//=============================================================================
// ST10_Flow7_CGlueing.scl
// 1:1 CONVERSION FROM TIA PORTAL V18 GRAPH XML
// Generated: 2026-02-02
//=============================================================================

TYPE
    E_STEP_ST10_Flow7_CGlueing : (
        STEP_ST10_Flow7_CGlueing_JudgeYPosition := 90,
        STEP_ST10_Flow7_CGlueing_CameraCheck1 := 118,
        STEP_ST10_Flow7_CGlueing_Step161 := 161,
        STEP_ST10_Flow7_CGlueing_Servo_returns_toGluePos_4 := 56,
        STEP_ST10_Flow7_CGlueing_OKStatus_3 := 135,
        STEP_ST10_Flow7_CGlueing_MESOverTime_1 := 318,
        STEP_ST10_Flow7_CGlueing_Axis_YToGlueePos_5 := 41,
        STEP_ST10_Flow7_CGlueing_ShaftGlueCameraCheck := 250,
        STEP_ST10_Flow7_CGlueing_CheckGlueSysOK_4 := 72,
        STEP_ST10_Flow7_CGlueing_ResetMesCheckRequest_1 := 302,
        STEP_ST10_Flow7_CGlueing_ServoHomePos_5 := 143,
        STEP_ST10_Flow7_CGlueing_MES_Check := 150,
        STEP_ST10_Flow7_CGlueing_Axis_XToGluePos_6 := 92,
        STEP_ST10_Flow7_CGlueing_Axis_ZToGlueePos_6 := 93,
        STEP_ST10_Flow7_CGlueing_CameraCheck4 := 137,
        STEP_ST10_Flow7_CGlueing_CheckIV3Ready_3 := 207,
        STEP_ST10_Flow7_CGlueing_Axis_XToGluePos_4 := 54,
        STEP_ST10_Flow7_CGlueing_GluePos_2 := 98,
        STEP_ST10_Flow7_CGlueing_OKStatus_4 := 141,
        STEP_ST10_Flow7_CGlueing_GlueFinishStatus := 83,
        STEP_ST10_Flow7_CGlueing_Axis_XToGluePos_5 := 71,
        STEP_ST10_Flow7_CGlueing_IAIMoveFinish_1 := 105,
        STEP_ST10_Flow7_CGlueing_MESOverTime := 323,
        STEP_ST10_Flow7_CGlueing_Axis_YToGluePos_6 := 91,
        STEP_ST10_Flow7_CGlueing_CheckServo_returns_toHome_Pos_5 := 99,
        STEP_ST10_Flow7_CGlueing_Step104 := 104,
        STEP_ST10_Flow7_CGlueing_OKStatus_2 := 129,
        STEP_ST10_Flow7_CGlueing_StatusAlarm := 24,
        STEP_ST10_Flow7_CGlueing_IV3Check_2 := 127,
        STEP_ST10_Flow7_CGlueing_WaitRobotFinishTask_2 := 289,
        STEP_ST10_Flow7_CGlueing_JudgeCheckStatus_3 := 134,
        STEP_ST10_Flow7_CGlueing_Axis_XToGluePos_2 := 36,
        STEP_ST10_Flow7_CGlueing_Axis_XToGlueSafPos_4 := 57,
        STEP_ST10_Flow7_CGlueing_PutMagnet := 64,
        STEP_ST10_Flow7_CGlueing_NGStatus_4 := 142,
        STEP_ST10_Flow7_CGlueing_F7_Initial := 1,
        STEP_ST10_Flow7_CGlueing_ok := 311,
        STEP_ST10_Flow7_CGlueing_Axis_ZToGlueePos_7 := 148,
        STEP_ST10_Flow7_CGlueing_CheckGlueSysOK_1 := 37,
        STEP_ST10_Flow7_CGlueing_ServoJoging := 123,
        STEP_ST10_Flow7_CGlueing_IAIMoveFinish_3 := 111,
        STEP_ST10_Flow7_CGlueing_RobotGluePick := 400,
        STEP_ST10_Flow7_CGlueing_C_LocationCylinderToHP2 := 122,
        STEP_ST10_Flow7_CGlueing_CheckIV3Ready_1 := 204,
        STEP_ST10_Flow7_CGlueing_Glue_3 := 50,
        STEP_ST10_Flow7_CGlueing_MES_Check_OK := 306,
        STEP_ST10_Flow7_CGlueing_Prepare_MES_CheckData := 303,
        STEP_ST10_Flow7_CGlueing_ServoHomePos_1 := 97,
        STEP_ST10_Flow7_CGlueing_Shaft_Glue := 287,
        STEP_ST10_Flow7_CGlueing_JudgeCheckStatus_4 := 140,
        STEP_ST10_Flow7_CGlueing_MESSaveRequest_1 := 313,
        STEP_ST10_Flow7_CGlueing_Axis_XYToHomePos_1 := 86,
        STEP_ST10_Flow7_CGlueing_JudgeCheckStatus := 61,
        STEP_ST10_Flow7_CGlueing_CameraCheck3 := 131,
        STEP_ST10_Flow7_CGlueing_Axis_ZToHomePos_2 := 82,
        STEP_ST10_Flow7_CGlueing_RequestRobotPutMagnet_1 := 281,
        STEP_ST10_Flow7_CGlueing_MESResult := 151,
        STEP_ST10_Flow7_CGlueing_CheckIV3Ready := 202,
        STEP_ST10_Flow7_CGlueing_MES__Check_Result := 350,
        STEP_ST10_Flow7_CGlueing_StopServoJoging := 124,
        STEP_ST10_Flow7_CGlueing_NGStatus := 63,
        STEP_ST10_Flow7_CGlueing_OKPart := 152,
        STEP_ST10_Flow7_CGlueing_IAIMoveFinish := 95,
        STEP_ST10_Flow7_CGlueing_Step159 := 159,
        STEP_ST10_Flow7_CGlueing_Step160 := 160,
        STEP_ST10_Flow7_CGlueing_Servo_returns_toGluePos_8 := 138,
        STEP_ST10_Flow7_CGlueing_Axis_YToGlueePos_1 := 26,
        STEP_ST10_Flow7_CGlueing_S10_InitialFinish := 10,
        STEP_ST10_Flow7_CGlueing_CheckIV3Ready_2 := 206,
        STEP_ST10_Flow7_CGlueing_Check_OK := 316,
        STEP_ST10_Flow7_CGlueing_NGStatus_3 := 136,
        STEP_ST10_Flow7_CGlueing_GluePos_1 := 96,
        STEP_ST10_Flow7_CGlueing_PartNG := 401,
        STEP_ST10_Flow7_CGlueing_JudgeCheckStatus_2 := 128,
        STEP_ST10_Flow7_CGlueing_RequestRobot1PutShaft := 27,
        STEP_ST10_Flow7_CGlueing_MES_Check_OK_1 := 399,
        STEP_ST10_Flow7_CGlueing_Process_Finish := 149,
        STEP_ST10_Flow7_CGlueing_Shaft_GlueCheck := 67,
        STEP_ST10_Flow7_CGlueing_ServoReady_ := 6,
        STEP_ST10_Flow7_CGlueing_MagnetGlueFinish := 349,
        STEP_ST10_Flow7_CGlueing_WaitRobotFinishTask_1 := 288,
        STEP_ST10_Flow7_CGlueing_Glue_2 := 40,
        STEP_ST10_Flow7_CGlueing_Bypass_1 := 324,
        STEP_ST10_Flow7_CGlueing_Step314 := 322,
        STEP_ST10_Flow7_CGlueing_Axis_ZToGlueePos_5 := 70,
        STEP_ST10_Flow7_CGlueing_IV3Check_1 := 69,
        STEP_ST10_Flow7_CGlueing_Step102 := 102,
        STEP_ST10_Flow7_CGlueing_Axis_YToGlueePos_7 := 88,
        STEP_ST10_Flow7_CGlueing_Servo_returns_toGluePos_2 := 38,
        STEP_ST10_Flow7_CGlueing_Axis_XToGluePos_3 := 46,
        STEP_ST10_Flow7_CGlueing_S4 := 4,
        STEP_ST10_Flow7_CGlueing_C_LocationCylinderToWP_1 := 120,
        STEP_ST10_Flow7_CGlueing_IAIMoveFinish__1 := 153,
        STEP_ST10_Flow7_CGlueing_JudgeCheckStatus_1 := 74,
        STEP_ST10_Flow7_CGlueing_Axis_ZToHomePos_1 := 80,
        STEP_ST10_Flow7_CGlueing_GluePos_4 := 116,
        STEP_ST10_Flow7_CGlueing_Axis_XToGlueSafPos_3 := 49,
        STEP_ST10_Flow7_CGlueing_ShaftGlueFinishStatus := 68,
        STEP_ST10_Flow7_CGlueing_Servo_returns_toGluePos_6 := 125,
        STEP_ST10_Flow7_CGlueing_Axis_XToHomePos := 81,
        STEP_ST10_Flow7_CGlueing_Step87 := 87,
        STEP_ST10_Flow7_CGlueing_Step315 := 328,
        STEP_ST10_Flow7_CGlueing_CheckPartStatus := 23,
        STEP_ST10_Flow7_CGlueing_Step158 := 158,
        STEP_ST10_Flow7_CGlueing_WaitIAIStop := 103,
        STEP_ST10_Flow7_CGlueing_Axis_ZToGlueePos_3 := 45,
        STEP_ST10_Flow7_CGlueing_CheckGlueSysOK_3 := 55,
        STEP_ST10_Flow7_CGlueing_WaitTableCode_OK := 101,
        STEP_ST10_Flow7_CGlueing_Axis_YToGlueePos_6 := 52,
        STEP_ST10_Flow7_CGlueing_NGStatus_1 := 85,
        STEP_ST10_Flow7_CGlueing_GluePos_3 := 114,
        STEP_ST10_Flow7_CGlueing_Step146 := 146,
        STEP_ST10_Flow7_CGlueing_Axis_XYToHomePos_2 := 156,
        STEP_ST10_Flow7_CGlueing_S3 := 3,
        STEP_ST10_Flow7_CGlueing_ServoHomePos_2 := 113,
        STEP_ST10_Flow7_CGlueing_Servo_returns_toGluePos_5 := 73,
        STEP_ST10_Flow7_CGlueing_ResetMesCheckRequest := 301,
        STEP_ST10_Flow7_CGlueing_Axis_XYIVCheckPos := 79,
        STEP_ST10_Flow7_CGlueing_OKStatus := 62,
        STEP_ST10_Flow7_CGlueing_S5_MESInitial := 5,
        STEP_ST10_Flow7_CGlueing_ShaftGluingProcess := 200,
        STEP_ST10_Flow7_CGlueing_Axis_ZToGlueePos_4 := 53,
        STEP_ST10_Flow7_CGlueing_CheckGlueSysOK_2 := 47,
        STEP_ST10_Flow7_CGlueing_RobotPutMagnet := 300,
        STEP_ST10_Flow7_CGlueing_TimeDelay_4 := 59,
        STEP_ST10_Flow7_CGlueing_Axis_XYIVCheckPos_1 := 157,
        STEP_ST10_Flow7_CGlueing_Axis_YToGluePos_5 := 75,
        STEP_ST10_Flow7_CGlueing_C_LocationCylinderToWP_2 := 121,
        STEP_ST10_Flow7_CGlueing_ServoHomePos_4 := 117,
        STEP_ST10_Flow7_CGlueing_Servo_returns_toGluePos_1 := 31,
        STEP_ST10_Flow7_CGlueing_ProcessStart := 100,
        STEP_ST10_Flow7_CGlueing_Servo_returns_toGluePos_7 := 132,
        STEP_ST10_Flow7_CGlueing_Axis_XToGlueSafPos_2 := 39,
        STEP_ST10_Flow7_CGlueing_TimeDelay_3 := 51,
        STEP_ST10_Flow7_CGlueing_ServoHomePos_6 := 144,
        STEP_ST10_Flow7_CGlueing_RequestRobotGluePick := 282,
        STEP_ST10_Flow7_CGlueing_MESCheckRequest := 310,
        STEP_ST10_Flow7_CGlueing_Axis_ZToIVCheckPos := 78,
        STEP_ST10_Flow7_CGlueing_ok_1 := 329,
        STEP_ST10_Flow7_CGlueing_CheckGlueSysOK := 30,
        STEP_ST10_Flow7_CGlueing_IAIMoveFinish_2 := 108,
        STEP_ST10_Flow7_CGlueing_Axis_ZToGlueePos_1 := 89,
        STEP_ST10_Flow7_CGlueing_Glue2s := 163,
        STEP_ST10_Flow7_CGlueing_ServoHomePos := 94,
        STEP_ST10_Flow7_CGlueing_Axis_ZToGlueePos_2 := 35,
        STEP_ST10_Flow7_CGlueing_IV3Check := 60,
        STEP_ST10_Flow7_CGlueing_Step110 := 110,
        STEP_ST10_Flow7_CGlueing_Magnet_Glue := 65,
        STEP_ST10_Flow7_CGlueing_Servo_returns_toGluePos_3 := 48,
        STEP_ST10_Flow7_CGlueing_WaitIAIStop_3 := 112,
        STEP_ST10_Flow7_CGlueing_ResultNG := 326,
        STEP_ST10_Flow7_CGlueing_NGStatus_2 := 130,
        STEP_ST10_Flow7_CGlueing_TimeDelay_1 := 42,
        STEP_ST10_Flow7_CGlueing_Bypass := 315,
        STEP_ST10_Flow7_CGlueing_IAIMoveFinish_4 := 155,
        STEP_ST10_Flow7_CGlueing_CheckIV3Ready_4 := 208,
        STEP_ST10_Flow7_CGlueing_ShaftGlueProcessFinish := 299,
        STEP_ST10_Flow7_CGlueing_WaitIAIStop_1 := 106,
        STEP_ST10_Flow7_CGlueing_Check_NG := 317,
        STEP_ST10_Flow7_CGlueing_TimeDelay_5 := 76,
        STEP_ST10_Flow7_CGlueing_Servo_returns_toHome_Pos := 22,
        STEP_ST10_Flow7_CGlueing_ServoHomePos_3 := 115,
        STEP_ST10_Flow7_CGlueing_CameraCheck2 := 126,
        STEP_ST10_Flow7_CGlueing_WaitRobot1FinishTask := 28,
        STEP_ST10_Flow7_CGlueing_bypassGlue4 := 162,
        STEP_ST10_Flow7_CGlueing_IV3Check_4 := 139,
        STEP_ST10_Flow7_CGlueing_IV3_Check := 630,
        STEP_ST10_Flow7_CGlueing_Prepare_MES_CheckData_1 := 307,
        STEP_ST10_Flow7_CGlueing_MaganetGlue := 320,
        STEP_ST10_Flow7_CGlueing_WaitIAIStop_2 := 109,
        STEP_ST10_Flow7_CGlueing_Axis_XToGlueSafPos := 32,
        STEP_ST10_Flow7_CGlueing_IAIMoveFinish_5 := 154,
        STEP_ST10_Flow7_CGlueing_Total_Score_of_Shaft_Gluening_check := 203,
        STEP_ST10_Flow7_CGlueing_Axis_YToHomePos := 21,
        STEP_ST10_Flow7_CGlueing_TimeDelay_2 := 43,
        STEP_ST10_Flow7_CGlueing_Step145 := 145,
        STEP_ST10_Flow7_CGlueing_CheckAxisXPos := 147,
        STEP_ST10_Flow7_CGlueing_C_LocationCylinderToHP := 119,
        STEP_ST10_Flow7_CGlueing_OKStatus_1 := 84,
        STEP_ST10_Flow7_CGlueing_Step204 := 205,
        STEP_ST10_Flow7_CGlueing_Step107 := 107,
        STEP_ST10_Flow7_CGlueing_Process__Finish := 290,
        STEP_ST10_Flow7_CGlueing_Glue_4 := 58,
        STEP_ST10_Flow7_CGlueing_Glue_1 := 33,
        STEP_ST10_Flow7_CGlueing_IV3Check_3 := 133,
        STEP_ST10_Flow7_CGlueing_Magnet_GlueCheck := 66,
        STEP_ST10_Flow7_CGlueing_WaitRobotInitialFinish := 8,
        STEP_ST10_Flow7_CGlueing_S2 := 2,
        STEP_ST10_Flow7_CGlueing_Axis_XToGluePos_1 := 29,
    ) INT := 1;
END_TYPE

CONST
    STEP_ST10_Flow7_CGlueing_JudgeYPosition := 90;
    STEP_ST10_Flow7_CGlueing_CameraCheck1 := 118;
    STEP_ST10_Flow7_CGlueing_Step161 := 161;
    STEP_ST10_Flow7_CGlueing_Servo_returns_toGluePos_4 := 56;
    STEP_ST10_Flow7_CGlueing_OKStatus_3 := 135;
    STEP_ST10_Flow7_CGlueing_MESOverTime_1 := 318;
    STEP_ST10_Flow7_CGlueing_Axis_YToGlueePos_5 := 41;
    STEP_ST10_Flow7_CGlueing_ShaftGlueCameraCheck := 250;
    STEP_ST10_Flow7_CGlueing_CheckGlueSysOK_4 := 72;
    STEP_ST10_Flow7_CGlueing_ResetMesCheckRequest_1 := 302;
    STEP_ST10_Flow7_CGlueing_ServoHomePos_5 := 143;
    STEP_ST10_Flow7_CGlueing_MES_Check := 150;
    STEP_ST10_Flow7_CGlueing_Axis_XToGluePos_6 := 92;
    STEP_ST10_Flow7_CGlueing_Axis_ZToGlueePos_6 := 93;
    STEP_ST10_Flow7_CGlueing_CameraCheck4 := 137;
    STEP_ST10_Flow7_CGlueing_CheckIV3Ready_3 := 207;
    STEP_ST10_Flow7_CGlueing_Axis_XToGluePos_4 := 54;
    STEP_ST10_Flow7_CGlueing_GluePos_2 := 98;
    STEP_ST10_Flow7_CGlueing_OKStatus_4 := 141;
    STEP_ST10_Flow7_CGlueing_GlueFinishStatus := 83;
    STEP_ST10_Flow7_CGlueing_Axis_XToGluePos_5 := 71;
    STEP_ST10_Flow7_CGlueing_IAIMoveFinish_1 := 105;
    STEP_ST10_Flow7_CGlueing_MESOverTime := 323;
    STEP_ST10_Flow7_CGlueing_Axis_YToGluePos_6 := 91;
    STEP_ST10_Flow7_CGlueing_CheckServo_returns_toHome_Pos_5 := 99;
    STEP_ST10_Flow7_CGlueing_Step104 := 104;
    STEP_ST10_Flow7_CGlueing_OKStatus_2 := 129;
    STEP_ST10_Flow7_CGlueing_StatusAlarm := 24;
    STEP_ST10_Flow7_CGlueing_IV3Check_2 := 127;
    STEP_ST10_Flow7_CGlueing_WaitRobotFinishTask_2 := 289;
    STEP_ST10_Flow7_CGlueing_JudgeCheckStatus_3 := 134;
    STEP_ST10_Flow7_CGlueing_Axis_XToGluePos_2 := 36;
    STEP_ST10_Flow7_CGlueing_Axis_XToGlueSafPos_4 := 57;
    STEP_ST10_Flow7_CGlueing_PutMagnet := 64;
    STEP_ST10_Flow7_CGlueing_NGStatus_4 := 142;
    STEP_ST10_Flow7_CGlueing_F7_Initial := 1;
    STEP_ST10_Flow7_CGlueing_ok := 311;
    STEP_ST10_Flow7_CGlueing_Axis_ZToGlueePos_7 := 148;
    STEP_ST10_Flow7_CGlueing_CheckGlueSysOK_1 := 37;
    STEP_ST10_Flow7_CGlueing_ServoJoging := 123;
    STEP_ST10_Flow7_CGlueing_IAIMoveFinish_3 := 111;
    STEP_ST10_Flow7_CGlueing_RobotGluePick := 400;
    STEP_ST10_Flow7_CGlueing_C_LocationCylinderToHP2 := 122;
    STEP_ST10_Flow7_CGlueing_CheckIV3Ready_1 := 204;
    STEP_ST10_Flow7_CGlueing_Glue_3 := 50;
    STEP_ST10_Flow7_CGlueing_MES_Check_OK := 306;
    STEP_ST10_Flow7_CGlueing_Prepare_MES_CheckData := 303;
    STEP_ST10_Flow7_CGlueing_ServoHomePos_1 := 97;
    STEP_ST10_Flow7_CGlueing_Shaft_Glue := 287;
    STEP_ST10_Flow7_CGlueing_JudgeCheckStatus_4 := 140;
    STEP_ST10_Flow7_CGlueing_MESSaveRequest_1 := 313;
    STEP_ST10_Flow7_CGlueing_Axis_XYToHomePos_1 := 86;
    STEP_ST10_Flow7_CGlueing_JudgeCheckStatus := 61;
    STEP_ST10_Flow7_CGlueing_CameraCheck3 := 131;
    STEP_ST10_Flow7_CGlueing_Axis_ZToHomePos_2 := 82;
    STEP_ST10_Flow7_CGlueing_RequestRobotPutMagnet_1 := 281;
    STEP_ST10_Flow7_CGlueing_MESResult := 151;
    STEP_ST10_Flow7_CGlueing_CheckIV3Ready := 202;
    STEP_ST10_Flow7_CGlueing_MES__Check_Result := 350;
    STEP_ST10_Flow7_CGlueing_StopServoJoging := 124;
    STEP_ST10_Flow7_CGlueing_NGStatus := 63;
    STEP_ST10_Flow7_CGlueing_OKPart := 152;
    STEP_ST10_Flow7_CGlueing_IAIMoveFinish := 95;
    STEP_ST10_Flow7_CGlueing_Step159 := 159;
    STEP_ST10_Flow7_CGlueing_Step160 := 160;
    STEP_ST10_Flow7_CGlueing_Servo_returns_toGluePos_8 := 138;
    STEP_ST10_Flow7_CGlueing_Axis_YToGlueePos_1 := 26;
    STEP_ST10_Flow7_CGlueing_S10_InitialFinish := 10;
    STEP_ST10_Flow7_CGlueing_CheckIV3Ready_2 := 206;
    STEP_ST10_Flow7_CGlueing_Check_OK := 316;
    STEP_ST10_Flow7_CGlueing_NGStatus_3 := 136;
    STEP_ST10_Flow7_CGlueing_GluePos_1 := 96;
    STEP_ST10_Flow7_CGlueing_PartNG := 401;
    STEP_ST10_Flow7_CGlueing_JudgeCheckStatus_2 := 128;
    STEP_ST10_Flow7_CGlueing_RequestRobot1PutShaft := 27;
    STEP_ST10_Flow7_CGlueing_MES_Check_OK_1 := 399;
    STEP_ST10_Flow7_CGlueing_Process_Finish := 149;
    STEP_ST10_Flow7_CGlueing_Shaft_GlueCheck := 67;
    STEP_ST10_Flow7_CGlueing_ServoReady_ := 6;
    STEP_ST10_Flow7_CGlueing_MagnetGlueFinish := 349;
    STEP_ST10_Flow7_CGlueing_WaitRobotFinishTask_1 := 288;
    STEP_ST10_Flow7_CGlueing_Glue_2 := 40;
    STEP_ST10_Flow7_CGlueing_Bypass_1 := 324;
    STEP_ST10_Flow7_CGlueing_Step314 := 322;
    STEP_ST10_Flow7_CGlueing_Axis_ZToGlueePos_5 := 70;
    STEP_ST10_Flow7_CGlueing_IV3Check_1 := 69;
    STEP_ST10_Flow7_CGlueing_Step102 := 102;
    STEP_ST10_Flow7_CGlueing_Axis_YToGlueePos_7 := 88;
    STEP_ST10_Flow7_CGlueing_Servo_returns_toGluePos_2 := 38;
    STEP_ST10_Flow7_CGlueing_Axis_XToGluePos_3 := 46;
    STEP_ST10_Flow7_CGlueing_S4 := 4;
    STEP_ST10_Flow7_CGlueing_C_LocationCylinderToWP_1 := 120;
    STEP_ST10_Flow7_CGlueing_IAIMoveFinish__1 := 153;
    STEP_ST10_Flow7_CGlueing_JudgeCheckStatus_1 := 74;
    STEP_ST10_Flow7_CGlueing_Axis_ZToHomePos_1 := 80;
    STEP_ST10_Flow7_CGlueing_GluePos_4 := 116;
    STEP_ST10_Flow7_CGlueing_Axis_XToGlueSafPos_3 := 49;
    STEP_ST10_Flow7_CGlueing_ShaftGlueFinishStatus := 68;
    STEP_ST10_Flow7_CGlueing_Servo_returns_toGluePos_6 := 125;
    STEP_ST10_Flow7_CGlueing_Axis_XToHomePos := 81;
    STEP_ST10_Flow7_CGlueing_Step87 := 87;
    STEP_ST10_Flow7_CGlueing_Step315 := 328;
    STEP_ST10_Flow7_CGlueing_CheckPartStatus := 23;
    STEP_ST10_Flow7_CGlueing_Step158 := 158;
    STEP_ST10_Flow7_CGlueing_WaitIAIStop := 103;
    STEP_ST10_Flow7_CGlueing_Axis_ZToGlueePos_3 := 45;
    STEP_ST10_Flow7_CGlueing_CheckGlueSysOK_3 := 55;
    STEP_ST10_Flow7_CGlueing_WaitTableCode_OK := 101;
    STEP_ST10_Flow7_CGlueing_Axis_YToGlueePos_6 := 52;
    STEP_ST10_Flow7_CGlueing_NGStatus_1 := 85;
    STEP_ST10_Flow7_CGlueing_GluePos_3 := 114;
    STEP_ST10_Flow7_CGlueing_Step146 := 146;
    STEP_ST10_Flow7_CGlueing_Axis_XYToHomePos_2 := 156;
    STEP_ST10_Flow7_CGlueing_S3 := 3;
    STEP_ST10_Flow7_CGlueing_ServoHomePos_2 := 113;
    STEP_ST10_Flow7_CGlueing_Servo_returns_toGluePos_5 := 73;
    STEP_ST10_Flow7_CGlueing_ResetMesCheckRequest := 301;
    STEP_ST10_Flow7_CGlueing_Axis_XYIVCheckPos := 79;
    STEP_ST10_Flow7_CGlueing_OKStatus := 62;
    STEP_ST10_Flow7_CGlueing_S5_MESInitial := 5;
    STEP_ST10_Flow7_CGlueing_ShaftGluingProcess := 200;
    STEP_ST10_Flow7_CGlueing_Axis_ZToGlueePos_4 := 53;
    STEP_ST10_Flow7_CGlueing_CheckGlueSysOK_2 := 47;
    STEP_ST10_Flow7_CGlueing_RobotPutMagnet := 300;
    STEP_ST10_Flow7_CGlueing_TimeDelay_4 := 59;
    STEP_ST10_Flow7_CGlueing_Axis_XYIVCheckPos_1 := 157;
    STEP_ST10_Flow7_CGlueing_Axis_YToGluePos_5 := 75;
    STEP_ST10_Flow7_CGlueing_C_LocationCylinderToWP_2 := 121;
    STEP_ST10_Flow7_CGlueing_ServoHomePos_4 := 117;
    STEP_ST10_Flow7_CGlueing_Servo_returns_toGluePos_1 := 31;
    STEP_ST10_Flow7_CGlueing_ProcessStart := 100;
    STEP_ST10_Flow7_CGlueing_Servo_returns_toGluePos_7 := 132;
    STEP_ST10_Flow7_CGlueing_Axis_XToGlueSafPos_2 := 39;
    STEP_ST10_Flow7_CGlueing_TimeDelay_3 := 51;
    STEP_ST10_Flow7_CGlueing_ServoHomePos_6 := 144;
    STEP_ST10_Flow7_CGlueing_RequestRobotGluePick := 282;
    STEP_ST10_Flow7_CGlueing_MESCheckRequest := 310;
    STEP_ST10_Flow7_CGlueing_Axis_ZToIVCheckPos := 78;
    STEP_ST10_Flow7_CGlueing_ok_1 := 329;
    STEP_ST10_Flow7_CGlueing_CheckGlueSysOK := 30;
    STEP_ST10_Flow7_CGlueing_IAIMoveFinish_2 := 108;
    STEP_ST10_Flow7_CGlueing_Axis_ZToGlueePos_1 := 89;
    STEP_ST10_Flow7_CGlueing_Glue2s := 163;
    STEP_ST10_Flow7_CGlueing_ServoHomePos := 94;
    STEP_ST10_Flow7_CGlueing_Axis_ZToGlueePos_2 := 35;
    STEP_ST10_Flow7_CGlueing_IV3Check := 60;
    STEP_ST10_Flow7_CGlueing_Step110 := 110;
    STEP_ST10_Flow7_CGlueing_Magnet_Glue := 65;
    STEP_ST10_Flow7_CGlueing_Servo_returns_toGluePos_3 := 48;
    STEP_ST10_Flow7_CGlueing_WaitIAIStop_3 := 112;
    STEP_ST10_Flow7_CGlueing_ResultNG := 326;
    STEP_ST10_Flow7_CGlueing_NGStatus_2 := 130;
    STEP_ST10_Flow7_CGlueing_TimeDelay_1 := 42;
    STEP_ST10_Flow7_CGlueing_Bypass := 315;
    STEP_ST10_Flow7_CGlueing_IAIMoveFinish_4 := 155;
    STEP_ST10_Flow7_CGlueing_CheckIV3Ready_4 := 208;
    STEP_ST10_Flow7_CGlueing_ShaftGlueProcessFinish := 299;
    STEP_ST10_Flow7_CGlueing_WaitIAIStop_1 := 106;
    STEP_ST10_Flow7_CGlueing_Check_NG := 317;
    STEP_ST10_Flow7_CGlueing_TimeDelay_5 := 76;
    STEP_ST10_Flow7_CGlueing_Servo_returns_toHome_Pos := 22;
    STEP_ST10_Flow7_CGlueing_ServoHomePos_3 := 115;
    STEP_ST10_Flow7_CGlueing_CameraCheck2 := 126;
    STEP_ST10_Flow7_CGlueing_WaitRobot1FinishTask := 28;
    STEP_ST10_Flow7_CGlueing_bypassGlue4 := 162;
    STEP_ST10_Flow7_CGlueing_IV3Check_4 := 139;
    STEP_ST10_Flow7_CGlueing_IV3_Check := 630;
    STEP_ST10_Flow7_CGlueing_Prepare_MES_CheckData_1 := 307;
    STEP_ST10_Flow7_CGlueing_MaganetGlue := 320;
    STEP_ST10_Flow7_CGlueing_WaitIAIStop_2 := 109;
    STEP_ST10_Flow7_CGlueing_Axis_XToGlueSafPos := 32;
    STEP_ST10_Flow7_CGlueing_IAIMoveFinish_5 := 154;
    STEP_ST10_Flow7_CGlueing_Total_Score_of_Shaft_Gluening_check := 203;
    STEP_ST10_Flow7_CGlueing_Axis_YToHomePos := 21;
    STEP_ST10_Flow7_CGlueing_TimeDelay_2 := 43;
    STEP_ST10_Flow7_CGlueing_Step145 := 145;
    STEP_ST10_Flow7_CGlueing_CheckAxisXPos := 147;
    STEP_ST10_Flow7_CGlueing_C_LocationCylinderToHP := 119;
    STEP_ST10_Flow7_CGlueing_OKStatus_1 := 84;
    STEP_ST10_Flow7_CGlueing_Step204 := 205;
    STEP_ST10_Flow7_CGlueing_Step107 := 107;
    STEP_ST10_Flow7_CGlueing_Process__Finish := 290;
    STEP_ST10_Flow7_CGlueing_Glue_4 := 58;
    STEP_ST10_Flow7_CGlueing_Glue_1 := 33;
    STEP_ST10_Flow7_CGlueing_IV3Check_3 := 133;
    STEP_ST10_Flow7_CGlueing_Magnet_GlueCheck := 66;
    STEP_ST10_Flow7_CGlueing_WaitRobotInitialFinish := 8;
    STEP_ST10_Flow7_CGlueing_S2 := 2;
    STEP_ST10_Flow7_CGlueing_Axis_XToGluePos_1 := 29;
END_CONST

FUNCTION_BLOCK "ST10_Flow7_CGlueing_1to1"
{ S7_Optimized_Access := 'TRUE' }
VERSION : 1.0

VAR_INPUT
    iSysInface : "RCS_SysComInterface_V1";
END_VAR

VAR_IN_OUT
    ioPM_Inface : "RCS_PMInterface_V1";
    ioStatus : Int;
END_VAR

VAR_OUTPUT
    oAlarmID : Int;
END_VAR

VAR
    State : INT := 1;
    act_InitialRun : Bool;
    act_InitialOK : Bool;
    act_WaitRunning : Bool;
    act_Running : Bool;
    act_ProcessComplete : Bool;
    act_ProcessStart : Bool;
    act_UnPause : Bool;
    bError : Bool;
    wErrorID : Word;
END_VAR

BEGIN
    //======================================================================
    // STATE MACHINE - Inline Transition Conditions
    //======================================================================

    CASE #State OF

        // ===========================================
        // STEP 90: JudgeYPosition
        // ===========================================
        STEP_ST10_Flow7_CGlueing_JudgeYPosition:
            // No actions in XML

            // Transition to next step: 118
            IF TRUE THEN  // Sequential transition - review XML for actual condition
                #State := STEP_ST10_Flow7_CGlueing_CameraCheck1;
            END_IF;

        // ===========================================
        // STEP 118: CameraCheck1
        // ===========================================
        STEP_ST10_Flow7_CGlueing_CameraCheck1:
            // No actions in XML

            // Transition to next step: 161
            IF TRUE THEN  // Sequential transition - review XML for actual condition
                #State := STEP_ST10_Flow7_CGlueing_Step161;
            END_IF;

        // ===========================================
        // STEP 161: Step161
        // ===========================================
        STEP_ST10_Flow7_CGlueing_Step161:
            // No actions in XML

            // Transition to next step: 56
            IF TRUE THEN  // Sequential transition - review XML for actual condition
                #State := STEP_ST10_Flow7_CGlueing_Servo_returns_toGluePos_4;
            END_IF;

        // ===========================================
        // STEP 56: Servo returns toGluePos_4
        // ===========================================
        STEP_ST10_Flow7_CGlueing_Servo_returns_toGluePos_4:
            // Action Qualifier=N
            // Token: "ServoV90_DeviceCtl".V90Servo[3].Point[5].Start
            "ServoV90_DeviceCtl".V90Servo[3].Point[5].Start;

            // Transition to next step: 135
            IF TRUE THEN  // Sequential transition - review XML for actual condition
                #State := STEP_ST10_Flow7_CGlueing_OKStatus_3;
            END_IF;

        // ===========================================
        // STEP 135: OKStatus_3
        // ===========================================
        STEP_ST10_Flow7_CGlueing_OKStatus_3:
            // Action Qualifier=N
            // Token: "AutoProcessData".C_Glue.PartStatus := 310
            "AutoProcessData".C_Glue.PartStatus := 310;
            // Action Qualifier=N
            // Token: "Station5UnLoadData"."PLC.ShaftGlueIVScore3" := "DB_KeyenceCheckerIV3".aDev[2].In.ToolResult[2].nToolMatchingRate
            "Station5UnLoadData"."PLC.ShaftGlueIVScore3" := "DB_KeyenceCheckerIV3".aDev[2].In.ToolResult[2].nToolMatchingRate;
            // Action Qualifier=N
            // Token: "AutoProcessData".C_Glue.IV3_ShaftScore_3 := "DB_KeyenceCheckerIV3".aDev[2].In.ToolResult[2].nToolMatchingRate
            "AutoProcessData".C_Glue.IV3_ShaftScore_3 := "DB_KeyenceCheckerIV3".aDev[2].In.ToolResult[2].nToolMatchingRate;

            // Transition to next step: 318
            IF TRUE THEN  // Sequential transition - review XML for actual condition
                #State := STEP_ST10_Flow7_CGlueing_MESOverTime_1;
            END_IF;

        // ===========================================
        // STEP 318: MESOverTime_1
        // ===========================================
        STEP_ST10_Flow7_CGlueing_MESOverTime_1:
            // Action Qualifier=S
            // Token: "ST10_DeviceError".MES_Error.CheckInCompOverTime_5
            "ST10_DeviceError".MES_Error.CheckInCompOverTime_5 := TRUE;

            // Transition to next step: 41
            IF TRUE THEN  // Sequential transition - review XML for actual condition
                #State := STEP_ST10_Flow7_CGlueing_Axis_YToGlueePos_5;
            END_IF;

        // ===========================================
        // STEP 41: Axis_YToGlueePos_5
        // ===========================================
        STEP_ST10_Flow7_CGlueing_Axis_YToGlueePos_5:
            // Action Qualifier=N
            // Token: "IAI_DeviceCtl".IAIServo[#Y_axis].Point[3].Start
            "IAI_DeviceCtl".IAIServo[#Y_axis].Point[3].Start;

            // Transition to next step: 250
            IF TRUE THEN  // Sequential transition - review XML for actual condition
                #State := STEP_ST10_Flow7_CGlueing_ShaftGlueCameraCheck;
            END_IF;

        // ===========================================
        // STEP 250: ShaftGlueCameraCheck
        // ===========================================
        STEP_ST10_Flow7_CGlueing_ShaftGlueCameraCheck:
            // No actions in XML

            // Transition to next step: 72
            IF TRUE THEN  // Sequential transition - review XML for actual condition
                #State := STEP_ST10_Flow7_CGlueing_CheckGlueSysOK_4;
            END_IF;

        // ===========================================
        // STEP 72: CheckGlueSysOK_4
        // ===========================================
        STEP_ST10_Flow7_CGlueing_CheckGlueSysOK_4:
            // No actions in XML

            // Transition to next step: 302
            IF TRUE THEN  // Sequential transition - review XML for actual condition
                #State := STEP_ST10_Flow7_CGlueing_ResetMesCheckRequest_1;
            END_IF;

        // ===========================================
        // STEP 302: ResetMesCheckRequest_1
        // ===========================================
        STEP_ST10_Flow7_CGlueing_ResetMesCheckRequest_1:
            // Action Qualifier=R
            // Token: "PLCtoMES"."PLC.Load_Station5ChickInReq"
            "PLCtoMES"."PLC.Load_Station5ChickInReq" := FALSE;
            // Action Qualifier=R
            // Token: "MEStoPLC"."MES.Load_Station5PartOK"
            "MEStoPLC"."MES.Load_Station5PartOK" := FALSE;
            // Action Qualifier=R
            // Token: "MEStoPLC"."MES.Load_Station5PartNG"
            "MEStoPLC"."MES.Load_Station5PartNG" := FALSE;
            // Action Qualifier=R
            // Token: "MEStoPLC"."MES.Load_Station5ReqMesDone"
            "MEStoPLC"."MES.Load_Station5ReqMesDone" := FALSE;
            // Action Qualifier=R
            // Token: "MEStoPLC"."MES.Unload_ResultsStored5OK"
            "MEStoPLC"."MES.Unload_ResultsStored5OK" := FALSE;
            // Action Qualifier=R
            // Token: "MEStoPLC"."MES.Unload_ResultsStored5ReqMesDone"
            "MEStoPLC"."MES.Unload_ResultsStored5ReqMesDone" := FALSE;

            // Transition to next step: 143
            IF TRUE THEN  // Sequential transition - review XML for actual condition
                #State := STEP_ST10_Flow7_CGlueing_ServoHomePos_5;
            END_IF;

        // ===========================================
        // STEP 143: ServoHomePos_5
        // ===========================================
        STEP_ST10_Flow7_CGlueing_ServoHomePos_5:
            // Action Qualifier=S
            // Token: "ServoV90_A3".IO.ioAutoHome
            "ServoV90_A3".IO.ioAutoHome := TRUE;

            // Transition to next step: 150
            IF TRUE THEN  // Sequential transition - review XML for actual condition
                #State := STEP_ST10_Flow7_CGlueing_MES_Check;
            END_IF;

        // ===========================================
        // STEP 150: MES Check
        // ===========================================
        STEP_ST10_Flow7_CGlueing_MES_Check:
            // No actions in XML

            // Transition to next step: 92
            IF TRUE THEN  // Sequential transition - review XML for actual condition
                #State := STEP_ST10_Flow7_CGlueing_Axis_XToGluePos_6;
            END_IF;

        // ===========================================
        // STEP 92: Axis_XToGluePos_6
        // ===========================================
        STEP_ST10_Flow7_CGlueing_Axis_XToGluePos_6:
            // Action Qualifier=N
            // Token: "IAI_DeviceCtl".IAIServo[#X_Axis].Point[7].Start
            "IAI_DeviceCtl".IAIServo[#X_Axis].Point[7].Start;

            // Transition to next step: 93
            IF TRUE THEN  // Sequential transition - review XML for actual condition
                #State := STEP_ST10_Flow7_CGlueing_Axis_ZToGlueePos_6;
            END_IF;

        // ===========================================
        // STEP 93: Axis_ZToGlueePos_6
        // ===========================================
        STEP_ST10_Flow7_CGlueing_Axis_ZToGlueePos_6:
            // Action Qualifier=N
            // Token: "IAI_DeviceCtl".IAIServo[#Z_Axis].Point[6].Start
            "IAI_DeviceCtl".IAIServo[#Z_Axis].Point[6].Start;

            // Transition to next step: 137
            IF TRUE THEN  // Sequential transition - review XML for actual condition
                #State := STEP_ST10_Flow7_CGlueing_CameraCheck4;
            END_IF;

        // ===========================================
        // STEP 137: CameraCheck4
        // ===========================================
        STEP_ST10_Flow7_CGlueing_CameraCheck4:
            // No actions in XML

            // Transition to next step: 207
            IF TRUE THEN  // Sequential transition - review XML for actual condition
                #State := STEP_ST10_Flow7_CGlueing_CheckIV3Ready_3;
            END_IF;

        // ===========================================
        // STEP 207: CheckIV3Ready_3
        // ===========================================
        STEP_ST10_Flow7_CGlueing_CheckIV3Ready_3:
            // Action Qualifier=N
            // Token: "DB_KeyenceCheckerIV3".aDev[2].Para.nProgramNo := 1
            "DB_KeyenceCheckerIV3".aDev[2].Para.nProgramNo := 1;

            // Transition to next step: 54
            IF TRUE THEN  // Sequential transition - review XML for actual condition
                #State := STEP_ST10_Flow7_CGlueing_Axis_XToGluePos_4;
            END_IF;

        // ===========================================
        // STEP 54: Axis_XToGluePos_4
        // ===========================================
        STEP_ST10_Flow7_CGlueing_Axis_XToGluePos_4:
            // Action Qualifier=N
            // Token: "IAI_DeviceCtl".IAIServo[#X_Axis].Point[6].Start
            "IAI_DeviceCtl".IAIServo[#X_Axis].Point[6].Start;

            // Transition to next step: 98
            IF TRUE THEN  // Sequential transition - review XML for actual condition
                #State := STEP_ST10_Flow7_CGlueing_GluePos_2;
            END_IF;

        // ===========================================
        // STEP 98: GluePos_2
        // ===========================================
        STEP_ST10_Flow7_CGlueing_GluePos_2:
            // No actions in XML

            // Transition to next step: 141
            IF TRUE THEN  // Sequential transition - review XML for actual condition
                #State := STEP_ST10_Flow7_CGlueing_OKStatus_4;
            END_IF;

        // ===========================================
        // STEP 141: OKStatus_4
        // ===========================================
        STEP_ST10_Flow7_CGlueing_OKStatus_4:
            // Action Qualifier=N
            // Token: "AutoProcessData".C_Glue.PartStatus := 310
            "AutoProcessData".C_Glue.PartStatus := 310;
            // Action Qualifier=N
            // Token: "Station5UnLoadData"."PLC.ShaftGlueIVScore4" := "DB_KeyenceCheckerIV3".aDev[2].In.ToolResult[2].nToolMatchingRate
            "Station5UnLoadData"."PLC.ShaftGlueIVScore4" := "DB_KeyenceCheckerIV3".aDev[2].In.ToolResult[2].nToolMatchingRate;
            // Action Qualifier=N
            // Token: "AutoProcessData".C_Glue.IV3_ShaftScore_4 := "DB_KeyenceCheckerIV3".aDev[2].In.ToolResult[2].nToolMatchingRate
            "AutoProcessData".C_Glue.IV3_ShaftScore_4 := "DB_KeyenceCheckerIV3".aDev[2].In.ToolResult[2].nToolMatchingRate;
            // Action Qualifier=N
            // Token: "AutoProcessData".C_Glue.IV3_ShaftCheckResult := 1
            "AutoProcessData".C_Glue.IV3_ShaftCheckResult := 1;

            // Transition to next step: 83
            IF TRUE THEN  // Sequential transition - review XML for actual condition
                #State := STEP_ST10_Flow7_CGlueing_GlueFinishStatus;
            END_IF;

        // ===========================================
        // STEP 83: GlueFinishStatus
        // ===========================================
        STEP_ST10_Flow7_CGlueing_GlueFinishStatus:
            // Action Qualifier=N
            // Token: "AutoProcessData".C_Glue.PartStatus := 330
            "AutoProcessData".C_Glue.PartStatus := 330;

            // Transition to next step: 71
            IF TRUE THEN  // Sequential transition - review XML for actual condition
                #State := STEP_ST10_Flow7_CGlueing_Axis_XToGluePos_5;
            END_IF;

        // ===========================================
        // STEP 71: Axis_XToGluePos_5
        // ===========================================
        STEP_ST10_Flow7_CGlueing_Axis_XToGluePos_5:
            // Action Qualifier=N
            // Token: "IAI_DeviceCtl".IAIServo[#X_Axis].Point[7].Start
            "IAI_DeviceCtl".IAIServo[#X_Axis].Point[7].Start;

            // Transition to next step: 105
            IF TRUE THEN  // Sequential transition - review XML for actual condition
                #State := STEP_ST10_Flow7_CGlueing_IAIMoveFinish_1;
            END_IF;

        // ===========================================
        // STEP 105: IAIMoveFinish_1
        // ===========================================
        STEP_ST10_Flow7_CGlueing_IAIMoveFinish_1:
            // No actions in XML

            // Transition to next step: 323
            IF TRUE THEN  // Sequential transition - review XML for actual condition
                #State := STEP_ST10_Flow7_CGlueing_MESOverTime;
            END_IF;

        // ===========================================
        // STEP 323: MESOverTime
        // ===========================================
        STEP_ST10_Flow7_CGlueing_MESOverTime:
            // Action Qualifier=S
            // Token: "ST10_DeviceError".MES_Error.CheckInResultOverTime_5
            "ST10_DeviceError".MES_Error.CheckInResultOverTime_5 := TRUE;

            // Transition to next step: 91
            IF TRUE THEN  // Sequential transition - review XML for actual condition
                #State := STEP_ST10_Flow7_CGlueing_Axis_YToGluePos_6;
            END_IF;

        // ===========================================
        // STEP 91: Axis_YToGluePos_6
        // ===========================================
        STEP_ST10_Flow7_CGlueing_Axis_YToGluePos_6:
            // Action Qualifier=N
            // Token: "IAI_DeviceCtl".IAIServo[#Y_axis].Point[6].Start
            "IAI_DeviceCtl".IAIServo[#Y_axis].Point[6].Start;

            // Transition to next step: 99
            IF TRUE THEN  // Sequential transition - review XML for actual condition
                #State := STEP_ST10_Flow7_CGlueing_CheckServo_returns_toHome_Pos_5;
            END_IF;

        // ===========================================
        // STEP 99: CheckServo returns toHome Pos_5
        // ===========================================
        STEP_ST10_Flow7_CGlueing_CheckServo_returns_toHome_Pos_5:
            // No actions in XML

            // Transition to next step: 104
            IF TRUE THEN  // Sequential transition - review XML for actual condition
                #State := STEP_ST10_Flow7_CGlueing_Step104;
            END_IF;

        // ===========================================
        // STEP 104: Step104
        // ===========================================
        STEP_ST10_Flow7_CGlueing_Step104:
            // No actions in XML

            // Transition to next step: 129
            IF TRUE THEN  // Sequential transition - review XML for actual condition
                #State := STEP_ST10_Flow7_CGlueing_OKStatus_2;
            END_IF;

        // ===========================================
        // STEP 129: OKStatus_2
        // ===========================================
        STEP_ST10_Flow7_CGlueing_OKStatus_2:
            // Action Qualifier=N
            // Token: "AutoProcessData".C_Glue.PartStatus := 310
            "AutoProcessData".C_Glue.PartStatus := 310;
            // Action Qualifier=N
            // Token: "Station5UnLoadData"."PLC.ShaftGlueIVScore2" := "DB_KeyenceCheckerIV3".aDev[2].In.ToolResult[2].nToolMatchingRate
            "Station5UnLoadData"."PLC.ShaftGlueIVScore2" := "DB_KeyenceCheckerIV3".aDev[2].In.ToolResult[2].nToolMatchingRate;
            // Action Qualifier=N
            // Token: "AutoProcessData".C_Glue.IV3_ShaftScore_2 := "DB_KeyenceCheckerIV3".aDev[2].In.ToolResult[2].nToolMatchingRate
            "AutoProcessData".C_Glue.IV3_ShaftScore_2 := "DB_KeyenceCheckerIV3".aDev[2].In.ToolResult[2].nToolMatchingRate;

            // Transition to next step: 24
            IF TRUE THEN  // Sequential transition - review XML for actual condition
                #State := STEP_ST10_Flow7_CGlueing_StatusAlarm;
            END_IF;

        // ===========================================
        // STEP 24: StatusAlarm
        // ===========================================
        STEP_ST10_Flow7_CGlueing_StatusAlarm:
            // Action Qualifier=S
            // Token: "ST10_DeviceError".C.CGlueing.StatusError
            "ST10_DeviceError".C.CGlueing.StatusError := TRUE;

            // Transition to next step: 127
            IF TRUE THEN  // Sequential transition - review XML for actual condition
                #State := STEP_ST10_Flow7_CGlueing_IV3Check_2;
            END_IF;

        // ===========================================
        // STEP 127: IV3Check_2
        // ===========================================
        STEP_ST10_Flow7_CGlueing_IV3Check_2:
            // Action Qualifier=N, Event="S1"
            // Token: "DB_KeyenceCheckerIV3".aDev[2].Common.nMode := 1
            "DB_KeyenceCheckerIV3".aDev[2].Common.nMode := 1;

            // Transition to next step: 289
            IF TRUE THEN  // Sequential transition - review XML for actual condition
                #State := STEP_ST10_Flow7_CGlueing_WaitRobotFinishTask_2;
            END_IF;

        // ===========================================
        // STEP 289: WaitRobotFinishTask_2
        // ===========================================
        STEP_ST10_Flow7_CGlueing_WaitRobotFinishTask_2:
            // No actions in XML

            // Transition to next step: 134
            IF TRUE THEN  // Sequential transition - review XML for actual condition
                #State := STEP_ST10_Flow7_CGlueing_JudgeCheckStatus_3;
            END_IF;

        // ===========================================
        // STEP 134: JudgeCheckStatus_3
        // ===========================================
        STEP_ST10_Flow7_CGlueing_JudgeCheckStatus_3:
            // No actions in XML

            // Transition to next step: 36
            IF TRUE THEN  // Sequential transition - review XML for actual condition
                #State := STEP_ST10_Flow7_CGlueing_Axis_XToGluePos_2;
            END_IF;

        // ===========================================
        // STEP 36: Axis_XToGluePos_2
        // ===========================================
        STEP_ST10_Flow7_CGlueing_Axis_XToGluePos_2:
            // Action Qualifier=N
            // Token: "IAI_DeviceCtl".IAIServo[#X_Axis].Point[4].Start
            "IAI_DeviceCtl".IAIServo[#X_Axis].Point[4].Start;

            // Transition to next step: 57
            IF TRUE THEN  // Sequential transition - review XML for actual condition
                #State := STEP_ST10_Flow7_CGlueing_Axis_XToGlueSafPos_4;
            END_IF;

        // ===========================================
        // STEP 57: Axis_XToGlueSafPos_4
        // ===========================================
        STEP_ST10_Flow7_CGlueing_Axis_XToGlueSafPos_4:
            // Action Qualifier=N
            // Token: "IAI_DeviceCtl".IAIServo[#X_Axis].Point[2].Start
            "IAI_DeviceCtl".IAIServo[#X_Axis].Point[2].Start;

            // Transition to next step: 64
            IF TRUE THEN  // Sequential transition - review XML for actual condition
                #State := STEP_ST10_Flow7_CGlueing_PutMagnet;
            END_IF;

        // ===========================================
        // STEP 64: PutMagnet
        // ===========================================
        STEP_ST10_Flow7_CGlueing_PutMagnet:
            // No actions in XML

            // Transition to next step: 142
            IF TRUE THEN  // Sequential transition - review XML for actual condition
                #State := STEP_ST10_Flow7_CGlueing_NGStatus_4;
            END_IF;

        // ===========================================
        // STEP 142: NGStatus_4
        // ===========================================
        STEP_ST10_Flow7_CGlueing_NGStatus_4:
            // Action Qualifier=N
            // Token: "AutoProcessData".C_Glue.PartStatus := 359
            "AutoProcessData".C_Glue.PartStatus := 359;
            // Action Qualifier=N
            // Token: "Station5UnLoadData"."PLC.ShaftGlueIVScore4" := "DB_KeyenceCheckerIV3".aDev[2].In.ToolResult[2].nToolMatchingRate
            "Station5UnLoadData"."PLC.ShaftGlueIVScore4" := "DB_KeyenceCheckerIV3".aDev[2].In.ToolResult[2].nToolMatchingRate;
            // Action Qualifier=N
            // Token: "AutoProcessData".C_Glue.IV3_ShaftScore_4 := "DB_KeyenceCheckerIV3".aDev[2].In.ToolResult[2].nToolMatchingRate
            "AutoProcessData".C_Glue.IV3_ShaftScore_4 := "DB_KeyenceCheckerIV3".aDev[2].In.ToolResult[2].nToolMatchingRate;
            // Action Qualifier=N
            // Token: "AutoProcessData".C_Glue.IV3_ShaftCheckResult := 2
            "AutoProcessData".C_Glue.IV3_ShaftCheckResult := 2;

            // Transition to next step: 1
            IF TRUE THEN  // Sequential transition - review XML for actual condition
                #State := STEP_ST10_Flow7_CGlueing_F7_Initial;
            END_IF;

        // ===========================================
        // STEP 1: F7_Initial
        // ===========================================
        STEP_ST10_Flow7_CGlueing_F7_Initial:
            // Action Qualifier=S
            // Token: #ioPM_Inface.InitialRun
            #ioPM_Inface.InitialRun := TRUE;
            // Action Qualifier=R
            // Token: #ioPM_Inface.InitialOK
            #ioPM_Inface.InitialOK := FALSE;
            // Action Qualifier=R
            // Token: #ioPM_Inface.WaitRunning
            #ioPM_Inface.WaitRunning := FALSE;
            // Action Qualifier=R
            // Token: #ioPM_Inface.Running
            #ioPM_Inface.Running := FALSE;
            // Action Qualifier=R
            // Token: #ioPM_Inface.UnPause
            #ioPM_Inface.UnPause := FALSE;
            // Action Qualifier=R
            // Token: "Station_Sys".Cmd.Calibration
            "Station_Sys".Cmd.Calibration := FALSE;
            // Action Qualifier=R
            // Token: "Station_Sys".Cmd.ChangeOver
            "Station_Sys".Cmd.ChangeOver := FALSE;
            // Action Qualifier=N
            // Token: //"ST350_Sys".Cmd.DryRun
            //"ST350_Sys".Cmd.DryRun;
            // Action Qualifier=R
            // Token: "Station_Sys".Cmd.Reserve
            "Station_Sys".Cmd.Reserve := FALSE;
            // Action Qualifier=R
            // Token: "Station_Sys".Cmd.OneCycle
            "Station_Sys".Cmd.OneCycle := FALSE;
            // Action Qualifier=R
            // Token: #ioPM_Inface.ProcessComplete
            #ioPM_Inface.ProcessComplete := FALSE;
            // Action Qualifier=R
            // Token: #ioPM_Inface.ProcessStart
            #ioPM_Inface.ProcessStart := FALSE;
            // Action Qualifier=R
            // Token: "AutoProcessControl".C_Glue.Robot1PutPrimit
            "AutoProcessControl".C_Glue.Robot1PutPrimit := FALSE;
            // Action Qualifier=R
            // Token: "AutoProcessControl".C_Glue.Robot2PickPrimit
            "AutoProcessControl".C_Glue.Robot2PickPrimit := FALSE;
            // Action Qualifier=R
            // Token: "AutoProcessControl".C_Glue.Robot2MaganePutPrimit
            "AutoProcessControl".C_Glue.Robot2MaganePutPrimit := FALSE;

            // Transition to next step: 311
            IF TRUE THEN  // Sequential transition - review XML for actual condition
                #State := STEP_ST10_Flow7_CGlueing_ok;
            END_IF;

        // ===========================================
        // STEP 311: ok
        // ===========================================
        STEP_ST10_Flow7_CGlueing_ok:
            // Action Qualifier=N
            // Token: "AutoProcessData".C_Glue.PartStatus := 399
            "AutoProcessData".C_Glue.PartStatus := 399;

            // Transition to next step: 148
            IF TRUE THEN  // Sequential transition - review XML for actual condition
                #State := STEP_ST10_Flow7_CGlueing_Axis_ZToGlueePos_7;
            END_IF;

        // ===========================================
        // STEP 148: Axis_ZToGlueePos_7
        // ===========================================
        STEP_ST10_Flow7_CGlueing_Axis_ZToGlueePos_7:
            // Action Qualifier=N
            // Token: "IAI_DeviceCtl".IAIServo[#Z_Axis].Point[9].Start
            "IAI_DeviceCtl".IAIServo[#Z_Axis].Point[9].Start;

            // Transition to next step: 37
            IF TRUE THEN  // Sequential transition - review XML for actual condition
                #State := STEP_ST10_Flow7_CGlueing_CheckGlueSysOK_1;
            END_IF;

        // ===========================================
        // STEP 37: CheckGlueSysOK_1
        // ===========================================
        STEP_ST10_Flow7_CGlueing_CheckGlueSysOK_1:
            // No actions in XML

            // Transition to next step: 123
            IF TRUE THEN  // Sequential transition - review XML for actual condition
                #State := STEP_ST10_Flow7_CGlueing_ServoJoging;
            END_IF;

        // ===========================================
        // STEP 123: ServoJoging
        // ===========================================
        STEP_ST10_Flow7_CGlueing_ServoJoging:
            // No actions in XML

            // Transition to next step: 111
            IF TRUE THEN  // Sequential transition - review XML for actual condition
                #State := STEP_ST10_Flow7_CGlueing_IAIMoveFinish_3;
            END_IF;

        // ===========================================
        // STEP 111: IAIMoveFinish_3
        // ===========================================
        STEP_ST10_Flow7_CGlueing_IAIMoveFinish_3:
            // No actions in XML

            // Transition to next step: 400
            IF TRUE THEN  // Sequential transition - review XML for actual condition
                #State := STEP_ST10_Flow7_CGlueing_RobotGluePick;
            END_IF;

        // ===========================================
        // STEP 400: RobotGluePick
        // ===========================================
        STEP_ST10_Flow7_CGlueing_RobotGluePick:
            // No actions in XML

            // Transition to next step: 122
            IF TRUE THEN  // Sequential transition - review XML for actual condition
                #State := STEP_ST10_Flow7_CGlueing_C_LocationCylinderToHP2;
            END_IF;

        // ===========================================
        // STEP 122: C-LocationCylinderToHP2
        // ===========================================
        STEP_ST10_Flow7_CGlueing_C_LocationCylinderToHP2:
            // Action Qualifier=S
            // Token: "ST10Cylinder".Cy[9].Inout.AutoGoHome
            "ST10Cylinder".Cy[9].Inout.AutoGoHome := TRUE;
            // Action Qualifier=R
            // Token: "ST10Cylinder".Cy[9].Inout.AutoGoWork
            "ST10Cylinder".Cy[9].Inout.AutoGoWork := FALSE;

            // Transition to next step: 204
            IF TRUE THEN  // Sequential transition - review XML for actual condition
                #State := STEP_ST10_Flow7_CGlueing_CheckIV3Ready_1;
            END_IF;

        // ===========================================
        // STEP 204: CheckIV3Ready_1
        // ===========================================
        STEP_ST10_Flow7_CGlueing_CheckIV3Ready_1:
            // Action Qualifier=N
            // Token: "DB_KeyenceCheckerIV3".aDev[1].Para.nProgramNo := 1
            "DB_KeyenceCheckerIV3".aDev[1].Para.nProgramNo := 1;

            // Transition to next step: 50
            IF TRUE THEN  // Sequential transition - review XML for actual condition
                #State := STEP_ST10_Flow7_CGlueing_Glue_3;
            END_IF;

        // ===========================================
        // STEP 50: Glue_3
        // ===========================================
        STEP_ST10_Flow7_CGlueing_Glue_3:
            // No actions in XML

            // Transition to next step: 306
            IF TRUE THEN  // Sequential transition - review XML for actual condition
                #State := STEP_ST10_Flow7_CGlueing_MES_Check_OK;
            END_IF;

        // ===========================================
        // STEP 306: MES Check OK
        // ===========================================
        STEP_ST10_Flow7_CGlueing_MES_Check_OK:
            // No actions in XML

            // Transition to next step: 303
            IF TRUE THEN  // Sequential transition - review XML for actual condition
                #State := STEP_ST10_Flow7_CGlueing_Prepare_MES_CheckData;
            END_IF;

        // ===========================================
        // STEP 303: Prepare MES CheckData
        // ===========================================
        STEP_ST10_Flow7_CGlueing_Prepare_MES_CheckData:
            // No actions in XML

            // Transition to next step: 97
            IF TRUE THEN  // Sequential transition - review XML for actual condition
                #State := STEP_ST10_Flow7_CGlueing_ServoHomePos_1;
            END_IF;

        // ===========================================
        // STEP 97: ServoHomePos_1
        // ===========================================
        STEP_ST10_Flow7_CGlueing_ServoHomePos_1:
            // Action Qualifier=S
            // Token: "ServoV90_A3".IO.ioAutoHome
            "ServoV90_A3".IO.ioAutoHome := TRUE;

            // Transition to next step: 287
            IF TRUE THEN  // Sequential transition - review XML for actual condition
                #State := STEP_ST10_Flow7_CGlueing_Shaft_Glue;
            END_IF;

        // ===========================================
        // STEP 287: Shaft Glue
        // ===========================================
        STEP_ST10_Flow7_CGlueing_Shaft_Glue:
            // No actions in XML

            // Transition to next step: 140
            IF TRUE THEN  // Sequential transition - review XML for actual condition
                #State := STEP_ST10_Flow7_CGlueing_JudgeCheckStatus_4;
            END_IF;

        // ===========================================
        // STEP 140: JudgeCheckStatus_4
        // ===========================================
        STEP_ST10_Flow7_CGlueing_JudgeCheckStatus_4:
            // No actions in XML

            // Transition to next step: 313
            IF TRUE THEN  // Sequential transition - review XML for actual condition
                #State := STEP_ST10_Flow7_CGlueing_MESSaveRequest_1;
            END_IF;

        // ===========================================
        // STEP 313: MESSaveRequest_1
        // ===========================================
        STEP_ST10_Flow7_CGlueing_MESSaveRequest_1:
            // Action Qualifier=N
            // Token: "PLCtoMES"."PLC.Unload_Station5DataSaveReq"
            "PLCtoMES"."PLC.Unload_Station5DataSaveReq";

            // Transition to next step: 86
            IF TRUE THEN  // Sequential transition - review XML for actual condition
                #State := STEP_ST10_Flow7_CGlueing_Axis_XYToHomePos_1;
            END_IF;

        // ===========================================
        // STEP 86: Axis_XYToHomePos_1
        // ===========================================
        STEP_ST10_Flow7_CGlueing_Axis_XYToHomePos_1:
            // Action Qualifier=N
            // Token: "IAI_DeviceCtl".IAIServo[#X_Axis].Point[1].Start
            "IAI_DeviceCtl".IAIServo[#X_Axis].Point[1].Start;

            // Transition to next step: 61
            IF TRUE THEN  // Sequential transition - review XML for actual condition
                #State := STEP_ST10_Flow7_CGlueing_JudgeCheckStatus;
            END_IF;

        // ===========================================
        // STEP 61: JudgeCheckStatus
        // ===========================================
        STEP_ST10_Flow7_CGlueing_JudgeCheckStatus:
            // No actions in XML

            // Transition to next step: 131
            IF TRUE THEN  // Sequential transition - review XML for actual condition
                #State := STEP_ST10_Flow7_CGlueing_CameraCheck3;
            END_IF;

        // ===========================================
        // STEP 131: CameraCheck3
        // ===========================================
        STEP_ST10_Flow7_CGlueing_CameraCheck3:
            // No actions in XML

            // Transition to next step: 82
            IF TRUE THEN  // Sequential transition - review XML for actual condition
                #State := STEP_ST10_Flow7_CGlueing_Axis_ZToHomePos_2;
            END_IF;

        // ===========================================
        // STEP 82: Axis_ZToHomePos_2
        // ===========================================
        STEP_ST10_Flow7_CGlueing_Axis_ZToHomePos_2:
            // Action Qualifier=N
            // Token: "IAI_DeviceCtl".IAIServo[#Z_Axis].Point[1].Start
            "IAI_DeviceCtl".IAIServo[#Z_Axis].Point[1].Start;

            // Transition to next step: 281
            IF TRUE THEN  // Sequential transition - review XML for actual condition
                #State := STEP_ST10_Flow7_CGlueing_RequestRobotPutMagnet_1;
            END_IF;

        // ===========================================
        // STEP 281: RequestRobotPutMagnet_1
        // ===========================================
        STEP_ST10_Flow7_CGlueing_RequestRobotPutMagnet_1:
            // Action Qualifier=N
            // Token: "AutoProcessControl".C_Glue.Robot2MaganePutPrimit
            "AutoProcessControl".C_Glue.Robot2MaganePutPrimit;

            // Transition to next step: 151
            IF TRUE THEN  // Sequential transition - review XML for actual condition
                #State := STEP_ST10_Flow7_CGlueing_MESResult;
            END_IF;

        // ===========================================
        // STEP 151: MESResult
        // ===========================================
        STEP_ST10_Flow7_CGlueing_MESResult:
            // No actions in XML

            // Transition to next step: 202
            IF TRUE THEN  // Sequential transition - review XML for actual condition
                #State := STEP_ST10_Flow7_CGlueing_CheckIV3Ready;
            END_IF;

        // ===========================================
        // STEP 202: CheckIV3Ready
        // ===========================================
        STEP_ST10_Flow7_CGlueing_CheckIV3Ready:
            // Action Qualifier=N
            // Token: "DB_KeyenceCheckerIV3".aDev[2].Para.nProgramNo := 1
            "DB_KeyenceCheckerIV3".aDev[2].Para.nProgramNo := 1;

            // Transition to next step: 350
            IF TRUE THEN  // Sequential transition - review XML for actual condition
                #State := STEP_ST10_Flow7_CGlueing_MES__Check_Result;
            END_IF;

        // ===========================================
        // STEP 350: MES  Check Result
        // ===========================================
        STEP_ST10_Flow7_CGlueing_MES__Check_Result:
            // No actions in XML

            // Transition to next step: 124
            IF TRUE THEN  // Sequential transition - review XML for actual condition
                #State := STEP_ST10_Flow7_CGlueing_StopServoJoging;
            END_IF;

        // ===========================================
        // STEP 124: StopServoJoging
        // ===========================================
        STEP_ST10_Flow7_CGlueing_StopServoJoging:
            // No actions in XML

            // Transition to next step: 63
            IF TRUE THEN  // Sequential transition - review XML for actual condition
                #State := STEP_ST10_Flow7_CGlueing_NGStatus;
            END_IF;

        // ===========================================
        // STEP 63: NGStatus
        // ===========================================
        STEP_ST10_Flow7_CGlueing_NGStatus:
            // Action Qualifier=N
            // Token: "AutoProcessData".C_Glue.PartStatus := 359
            "AutoProcessData".C_Glue.PartStatus := 359;
            // Action Qualifier=N
            // Token: "Station5UnLoadData"."PLC.ShaftGlueIVScore1" := "DB_KeyenceCheckerIV3".aDev[2].In.ToolResult[2].nToolMatchingRate
            "Station5UnLoadData"."PLC.ShaftGlueIVScore1" := "DB_KeyenceCheckerIV3".aDev[2].In.ToolResult[2].nToolMatchingRate;
            // Action Qualifier=N
            // Token: "AutoProcessData".C_Glue.IV3_ShaftScore_1 := "DB_KeyenceCheckerIV3".aDev[2].In.ToolResult[2].nToolMatchingRate
            "AutoProcessData".C_Glue.IV3_ShaftScore_1 := "DB_KeyenceCheckerIV3".aDev[2].In.ToolResult[2].nToolMatchingRate;
            // Action Qualifier=N
            // Token: "AutoProcessData".C_Glue.IV3_ShaftCheckResult := 2
            "AutoProcessData".C_Glue.IV3_ShaftCheckResult := 2;

            // Transition to next step: 152
            IF TRUE THEN  // Sequential transition - review XML for actual condition
                #State := STEP_ST10_Flow7_CGlueing_OKPart;
            END_IF;

        // ===========================================
        // STEP 152: OKPart
        // ===========================================
        STEP_ST10_Flow7_CGlueing_OKPart:
            // No actions in XML

            // Transition to next step: 95
            IF TRUE THEN  // Sequential transition - review XML for actual condition
                #State := STEP_ST10_Flow7_CGlueing_IAIMoveFinish;
            END_IF;

        // ===========================================
        // STEP 95: IAIMoveFinish
        // ===========================================
        STEP_ST10_Flow7_CGlueing_IAIMoveFinish:
            // No actions in XML

            // Transition to next step: 159
            IF TRUE THEN  // Sequential transition - review XML for actual condition
                #State := STEP_ST10_Flow7_CGlueing_Step159;
            END_IF;

        // ===========================================
        // STEP 159: Step159
        // ===========================================
        STEP_ST10_Flow7_CGlueing_Step159:
            // No actions in XML

            // Transition to next step: 160
            IF TRUE THEN  // Sequential transition - review XML for actual condition
                #State := STEP_ST10_Flow7_CGlueing_Step160;
            END_IF;

        // ===========================================
        // STEP 160: Step160
        // ===========================================
        STEP_ST10_Flow7_CGlueing_Step160:
            // No actions in XML

            // Transition to next step: 138
            IF TRUE THEN  // Sequential transition - review XML for actual condition
                #State := STEP_ST10_Flow7_CGlueing_Servo_returns_toGluePos_8;
            END_IF;

        // ===========================================
        // STEP 138: Servo returns toGluePos_8
        // ===========================================
        STEP_ST10_Flow7_CGlueing_Servo_returns_toGluePos_8:
            // Action Qualifier=N
            // Token: "ServoV90_DeviceCtl".V90Servo[3].Point[9].Start
            "ServoV90_DeviceCtl".V90Servo[3].Point[9].Start;

            // Transition to next step: 26
            IF TRUE THEN  // Sequential transition - review XML for actual condition
                #State := STEP_ST10_Flow7_CGlueing_Axis_YToGlueePos_1;
            END_IF;

        // ===========================================
        // STEP 26: Axis_YToGlueePos_1
        // ===========================================
        STEP_ST10_Flow7_CGlueing_Axis_YToGlueePos_1:
            // Action Qualifier=N
            // Token: "IAI_DeviceCtl".IAIServo[#Y_axis].Point[2].Start
            "IAI_DeviceCtl".IAIServo[#Y_axis].Point[2].Start;

            // Transition to next step: 10
            IF TRUE THEN  // Sequential transition - review XML for actual condition
                #State := STEP_ST10_Flow7_CGlueing_S10_InitialFinish;
            END_IF;

        // ===========================================
        // STEP 10: S10_InitialFinish
        // ===========================================
        STEP_ST10_Flow7_CGlueing_S10_InitialFinish:
            // Action Qualifier=S
            // Token: #ioPM_Inface.InitialOK
            #ioPM_Inface.InitialOK := TRUE;

            // Transition to next step: 206
            IF TRUE THEN  // Sequential transition - review XML for actual condition
                #State := STEP_ST10_Flow7_CGlueing_CheckIV3Ready_2;
            END_IF;

        // ===========================================
        // STEP 206: CheckIV3Ready_2
        // ===========================================
        STEP_ST10_Flow7_CGlueing_CheckIV3Ready_2:
            // Action Qualifier=N
            // Token: "DB_KeyenceCheckerIV3".aDev[2].Para.nProgramNo := 1
            "DB_KeyenceCheckerIV3".aDev[2].Para.nProgramNo := 1;

            // Transition to next step: 316
            IF TRUE THEN  // Sequential transition - review XML for actual condition
                #State := STEP_ST10_Flow7_CGlueing_Check_OK;
            END_IF;

        // ===========================================
        // STEP 316: Check OK
        // ===========================================
        STEP_ST10_Flow7_CGlueing_Check_OK:
            // No actions in XML

            // Transition to next step: 136
            IF TRUE THEN  // Sequential transition - review XML for actual condition
                #State := STEP_ST10_Flow7_CGlueing_NGStatus_3;
            END_IF;

        // ===========================================
        // STEP 136: NGStatus_3
        // ===========================================
        STEP_ST10_Flow7_CGlueing_NGStatus_3:
            // Action Qualifier=N
            // Token: "AutoProcessData".C_Glue.PartStatus := 359
            "AutoProcessData".C_Glue.PartStatus := 359;
            // Action Qualifier=N
            // Token: "Station5UnLoadData"."PLC.ShaftGlueIVScore3" := "DB_KeyenceCheckerIV3".aDev[2].In.ToolResult[2].nToolMatchingRate
            "Station5UnLoadData"."PLC.ShaftGlueIVScore3" := "DB_KeyenceCheckerIV3".aDev[2].In.ToolResult[2].nToolMatchingRate;
            // Action Qualifier=N
            // Token: "AutoProcessData".C_Glue.IV3_ShaftScore_3 := "DB_KeyenceCheckerIV3".aDev[2].In.ToolResult[2].nToolMatchingRate
            "AutoProcessData".C_Glue.IV3_ShaftScore_3 := "DB_KeyenceCheckerIV3".aDev[2].In.ToolResult[2].nToolMatchingRate;
            // Action Qualifier=N
            // Token: "AutoProcessData".C_Glue.IV3_ShaftCheckResult := 2
            "AutoProcessData".C_Glue.IV3_ShaftCheckResult := 2;

            // Transition to next step: 96
            IF TRUE THEN  // Sequential transition - review XML for actual condition
                #State := STEP_ST10_Flow7_CGlueing_GluePos_1;
            END_IF;

        // ===========================================
        // STEP 96: GluePos_1
        // ===========================================
        STEP_ST10_Flow7_CGlueing_GluePos_1:
            // No actions in XML

            // Transition to next step: 401
            IF TRUE THEN  // Sequential transition - review XML for actual condition
                #State := STEP_ST10_Flow7_CGlueing_PartNG;
            END_IF;

        // ===========================================
        // STEP 401: PartNG
        // ===========================================
        STEP_ST10_Flow7_CGlueing_PartNG:
            // No actions in XML

            // Transition to next step: 128
            IF TRUE THEN  // Sequential transition - review XML for actual condition
                #State := STEP_ST10_Flow7_CGlueing_JudgeCheckStatus_2;
            END_IF;

        // ===========================================
        // STEP 128: JudgeCheckStatus_2
        // ===========================================
        STEP_ST10_Flow7_CGlueing_JudgeCheckStatus_2:
            // No actions in XML

            // Transition to next step: 27
            IF TRUE THEN  // Sequential transition - review XML for actual condition
                #State := STEP_ST10_Flow7_CGlueing_RequestRobot1PutShaft;
            END_IF;

        // ===========================================
        // STEP 27: RequestRobot1PutShaft
        // ===========================================
        STEP_ST10_Flow7_CGlueing_RequestRobot1PutShaft:
            // Action Qualifier=N
            // Token: "AutoProcessControl".C_Glue.Robot1PutPrimit
            "AutoProcessControl".C_Glue.Robot1PutPrimit;

            // Transition to next step: 399
            IF TRUE THEN  // Sequential transition - review XML for actual condition
                #State := STEP_ST10_Flow7_CGlueing_MES_Check_OK_1;
            END_IF;

        // ===========================================
        // STEP 399: MES Check OK_1
        // ===========================================
        STEP_ST10_Flow7_CGlueing_MES_Check_OK_1:
            // No actions in XML

            // Transition to next step: 149
            IF TRUE THEN  // Sequential transition - review XML for actual condition
                #State := STEP_ST10_Flow7_CGlueing_Process_Finish;
            END_IF;

        // ===========================================
        // STEP 149: Process Finish
        // ===========================================
        STEP_ST10_Flow7_CGlueing_Process_Finish:
            // No actions in XML

            // Transition to next step: 67
            IF TRUE THEN  // Sequential transition - review XML for actual condition
                #State := STEP_ST10_Flow7_CGlueing_Shaft_GlueCheck;
            END_IF;

        // ===========================================
        // STEP 67: Shaft GlueCheck
        // ===========================================
        STEP_ST10_Flow7_CGlueing_Shaft_GlueCheck:
            // No actions in XML

            // Transition to next step: 6
            IF TRUE THEN  // Sequential transition - review XML for actual condition
                #State := STEP_ST10_Flow7_CGlueing_ServoReady_;
            END_IF;

        // ===========================================
        // STEP 6: ServoReady?
        // ===========================================
        STEP_ST10_Flow7_CGlueing_ServoReady_:
            // No actions in XML

            // Transition to next step: 349
            IF TRUE THEN  // Sequential transition - review XML for actual condition
                #State := STEP_ST10_Flow7_CGlueing_MagnetGlueFinish;
            END_IF;

        // ===========================================
        // STEP 349: MagnetGlueFinish
        // ===========================================
        STEP_ST10_Flow7_CGlueing_MagnetGlueFinish:
            // No actions in XML

            // Transition to next step: 288
            IF TRUE THEN  // Sequential transition - review XML for actual condition
                #State := STEP_ST10_Flow7_CGlueing_WaitRobotFinishTask_1;
            END_IF;

        // ===========================================
        // STEP 288: WaitRobotFinishTask_1
        // ===========================================
        STEP_ST10_Flow7_CGlueing_WaitRobotFinishTask_1:
            // No actions in XML

            // Transition to next step: 40
            IF TRUE THEN  // Sequential transition - review XML for actual condition
                #State := STEP_ST10_Flow7_CGlueing_Glue_2;
            END_IF;

        // ===========================================
        // STEP 40: Glue_2
        // ===========================================
        STEP_ST10_Flow7_CGlueing_Glue_2:
            // No actions in XML

            // Transition to next step: 324
            IF TRUE THEN  // Sequential transition - review XML for actual condition
                #State := STEP_ST10_Flow7_CGlueing_Bypass_1;
            END_IF;

        // ===========================================
        // STEP 324: Bypass_1
        // ===========================================
        STEP_ST10_Flow7_CGlueing_Bypass_1:
            // No actions in XML

            // Transition to next step: 322
            IF TRUE THEN  // Sequential transition - review XML for actual condition
                #State := STEP_ST10_Flow7_CGlueing_Step314;
            END_IF;

        // ===========================================
        // STEP 322: Step314
        // ===========================================
        STEP_ST10_Flow7_CGlueing_Step314:
            // No actions in XML

            // Transition to next step: 70
            IF TRUE THEN  // Sequential transition - review XML for actual condition
                #State := STEP_ST10_Flow7_CGlueing_Axis_ZToGlueePos_5;
            END_IF;

        // ===========================================
        // STEP 70: Axis_ZToGlueePos_5
        // ===========================================
        STEP_ST10_Flow7_CGlueing_Axis_ZToGlueePos_5:
            // Action Qualifier=N
            // Token: "IAI_DeviceCtl".IAIServo[#Z_Axis].Point[6].Start
            "IAI_DeviceCtl".IAIServo[#Z_Axis].Point[6].Start;

            // Transition to next step: 69
            IF TRUE THEN  // Sequential transition - review XML for actual condition
                #State := STEP_ST10_Flow7_CGlueing_IV3Check_1;
            END_IF;

        // ===========================================
        // STEP 69: IV3Check_1
        // ===========================================
        STEP_ST10_Flow7_CGlueing_IV3Check_1:
            // Action Qualifier=N, Event="S1"
            // Token: "DB_KeyenceCheckerIV3".aDev[1].Common.nMode := 1
            "DB_KeyenceCheckerIV3".aDev[1].Common.nMode := 1;

            // Transition to next step: 102
            IF TRUE THEN  // Sequential transition - review XML for actual condition
                #State := STEP_ST10_Flow7_CGlueing_Step102;
            END_IF;

        // ===========================================
        // STEP 102: Step102
        // ===========================================
        STEP_ST10_Flow7_CGlueing_Step102:
            // No actions in XML

            // Transition to next step: 88
            IF TRUE THEN  // Sequential transition - review XML for actual condition
                #State := STEP_ST10_Flow7_CGlueing_Axis_YToGlueePos_7;
            END_IF;

        // ===========================================
        // STEP 88: Axis_YToGlueePos_7
        // ===========================================
        STEP_ST10_Flow7_CGlueing_Axis_YToGlueePos_7:
            // Action Qualifier=N
            // Token: "IAI_DeviceCtl".IAIServo[#Y_axis].Point[5].Start
            "IAI_DeviceCtl".IAIServo[#Y_axis].Point[5].Start;

            // Transition to next step: 38
            IF TRUE THEN  // Sequential transition - review XML for actual condition
                #State := STEP_ST10_Flow7_CGlueing_Servo_returns_toGluePos_2;
            END_IF;

        // ===========================================
        // STEP 38: Servo returns toGluePos_2
        // ===========================================
        STEP_ST10_Flow7_CGlueing_Servo_returns_toGluePos_2:
            // Action Qualifier=N
            // Token: "ServoV90_DeviceCtl".V90Servo[3].Point[3].Start
            "ServoV90_DeviceCtl".V90Servo[3].Point[3].Start;

            // Transition to next step: 46
            IF TRUE THEN  // Sequential transition - review XML for actual condition
                #State := STEP_ST10_Flow7_CGlueing_Axis_XToGluePos_3;
            END_IF;

        // ===========================================
        // STEP 46: Axis_XToGluePos_3
        // ===========================================
        STEP_ST10_Flow7_CGlueing_Axis_XToGluePos_3:
            // Action Qualifier=N
            // Token: "IAI_DeviceCtl".IAIServo[#X_Axis].Point[5].Start
            "IAI_DeviceCtl".IAIServo[#X_Axis].Point[5].Start;

            // Transition to next step: 4
            IF TRUE THEN  // Sequential transition - review XML for actual condition
                #State := STEP_ST10_Flow7_CGlueing_S4;
            END_IF;

        // ===========================================
        // STEP 4: S4
        // ===========================================
        STEP_ST10_Flow7_CGlueing_S4:
            // No actions in XML

            // Transition to next step: 120
            IF TRUE THEN  // Sequential transition - review XML for actual condition
                #State := STEP_ST10_Flow7_CGlueing_C_LocationCylinderToWP_1;
            END_IF;

        // ===========================================
        // STEP 120: C-LocationCylinderToWP_1
        // ===========================================
        STEP_ST10_Flow7_CGlueing_C_LocationCylinderToWP_1:
            // Action Qualifier=R
            // Token: "ST10Cylinder".Cy[9].Inout.AutoGoHome
            "ST10Cylinder".Cy[9].Inout.AutoGoHome := FALSE;
            // Action Qualifier=S
            // Token: "ST10Cylinder".Cy[9].Inout.AutoGoWork
            "ST10Cylinder".Cy[9].Inout.AutoGoWork := TRUE;

            // Transition to next step: 153
            IF TRUE THEN  // Sequential transition - review XML for actual condition
                #State := STEP_ST10_Flow7_CGlueing_IAIMoveFinish__1;
            END_IF;

        // ===========================================
        // STEP 153: IAIMoveFinish_ 1
        // ===========================================
        STEP_ST10_Flow7_CGlueing_IAIMoveFinish__1:
            // No actions in XML

            // Transition to next step: 74
            IF TRUE THEN  // Sequential transition - review XML for actual condition
                #State := STEP_ST10_Flow7_CGlueing_JudgeCheckStatus_1;
            END_IF;

        // ===========================================
        // STEP 74: JudgeCheckStatus_1
        // ===========================================
        STEP_ST10_Flow7_CGlueing_JudgeCheckStatus_1:
            // No actions in XML

            // Transition to next step: 80
            IF TRUE THEN  // Sequential transition - review XML for actual condition
                #State := STEP_ST10_Flow7_CGlueing_Axis_ZToHomePos_1;
            END_IF;

        // ===========================================
        // STEP 80: Axis_ZToHomePos_1
        // ===========================================
        STEP_ST10_Flow7_CGlueing_Axis_ZToHomePos_1:
            // Action Qualifier=N
            // Token: "IAI_DeviceCtl".IAIServo[#Z_Axis].Point[1].Start
            "IAI_DeviceCtl".IAIServo[#Z_Axis].Point[1].Start;

            // Transition to next step: 116
            IF TRUE THEN  // Sequential transition - review XML for actual condition
                #State := STEP_ST10_Flow7_CGlueing_GluePos_4;
            END_IF;

        // ===========================================
        // STEP 116: GluePos_4
        // ===========================================
        STEP_ST10_Flow7_CGlueing_GluePos_4:
            // No actions in XML

            // Transition to next step: 49
            IF TRUE THEN  // Sequential transition - review XML for actual condition
                #State := STEP_ST10_Flow7_CGlueing_Axis_XToGlueSafPos_3;
            END_IF;

        // ===========================================
        // STEP 49: Axis_XToGlueSafPos_3
        // ===========================================
        STEP_ST10_Flow7_CGlueing_Axis_XToGlueSafPos_3:
            // Action Qualifier=N
            // Token: "IAI_DeviceCtl".IAIServo[#X_Axis].Point[2].Start
            "IAI_DeviceCtl".IAIServo[#X_Axis].Point[2].Start;

            // Transition to next step: 68
            IF TRUE THEN  // Sequential transition - review XML for actual condition
                #State := STEP_ST10_Flow7_CGlueing_ShaftGlueFinishStatus;
            END_IF;

        // ===========================================
        // STEP 68: ShaftGlueFinishStatus
        // ===========================================
        STEP_ST10_Flow7_CGlueing_ShaftGlueFinishStatus:
            // Action Qualifier=N
            // Token: "AutoProcessData".C_Glue.PartStatus := 300
            "AutoProcessData".C_Glue.PartStatus := 300;

            // Transition to next step: 125
            IF TRUE THEN  // Sequential transition - review XML for actual condition
                #State := STEP_ST10_Flow7_CGlueing_Servo_returns_toGluePos_6;
            END_IF;

        // ===========================================
        // STEP 125: Servo returns toGluePos_6
        // ===========================================
        STEP_ST10_Flow7_CGlueing_Servo_returns_toGluePos_6:
            // Action Qualifier=N
            // Token: "ServoV90_DeviceCtl".V90Servo[3].Point[7].Start
            "ServoV90_DeviceCtl".V90Servo[3].Point[7].Start;

            // Transition to next step: 81
            IF TRUE THEN  // Sequential transition - review XML for actual condition
                #State := STEP_ST10_Flow7_CGlueing_Axis_XToHomePos;
            END_IF;

        // ===========================================
        // STEP 81: Axis_XToHomePos
        // ===========================================
        STEP_ST10_Flow7_CGlueing_Axis_XToHomePos:
            // Action Qualifier=N
            // Token: "IAI_DeviceCtl".IAIServo[#X_Axis].Point[1].Start
            "IAI_DeviceCtl".IAIServo[#X_Axis].Point[1].Start;

            // Transition to next step: 87
            IF TRUE THEN  // Sequential transition - review XML for actual condition
                #State := STEP_ST10_Flow7_CGlueing_Step87;
            END_IF;

        // ===========================================
        // STEP 87: Step87
        // ===========================================
        STEP_ST10_Flow7_CGlueing_Step87:
            // No actions in XML

            // Transition to next step: 328
            IF TRUE THEN  // Sequential transition - review XML for actual condition
                #State := STEP_ST10_Flow7_CGlueing_Step315;
            END_IF;

        // ===========================================
        // STEP 328: Step315
        // ===========================================
        STEP_ST10_Flow7_CGlueing_Step315:
            // No actions in XML

            // Transition to next step: 23
            IF TRUE THEN  // Sequential transition - review XML for actual condition
                #State := STEP_ST10_Flow7_CGlueing_CheckPartStatus;
            END_IF;

        // ===========================================
        // STEP 23: CheckPartStatus
        // ===========================================
        STEP_ST10_Flow7_CGlueing_CheckPartStatus:
            // No actions in XML

            // Transition to next step: 158
            IF TRUE THEN  // Sequential transition - review XML for actual condition
                #State := STEP_ST10_Flow7_CGlueing_Step158;
            END_IF;

        // ===========================================
        // STEP 158: Step158
        // ===========================================
        STEP_ST10_Flow7_CGlueing_Step158:
            // No actions in XML

            // Transition to next step: 103
            IF TRUE THEN  // Sequential transition - review XML for actual condition
                #State := STEP_ST10_Flow7_CGlueing_WaitIAIStop;
            END_IF;

        // ===========================================
        // STEP 103: WaitIAIStop
        // ===========================================
        STEP_ST10_Flow7_CGlueing_WaitIAIStop:
            // No actions in XML

            // Transition to next step: 45
            IF TRUE THEN  // Sequential transition - review XML for actual condition
                #State := STEP_ST10_Flow7_CGlueing_Axis_ZToGlueePos_3;
            END_IF;

        // ===========================================
        // STEP 45: Axis_ZToGlueePos_3
        // ===========================================
        STEP_ST10_Flow7_CGlueing_Axis_ZToGlueePos_3:
            // Action Qualifier=N
            // Token: "IAI_DeviceCtl".IAIServo[#Z_Axis].Point[4].Start
            "IAI_DeviceCtl".IAIServo[#Z_Axis].Point[4].Start;

            // Transition to next step: 55
            IF TRUE THEN  // Sequential transition - review XML for actual condition
                #State := STEP_ST10_Flow7_CGlueing_CheckGlueSysOK_3;
            END_IF;

        // ===========================================
        // STEP 55: CheckGlueSysOK_3
        // ===========================================
        STEP_ST10_Flow7_CGlueing_CheckGlueSysOK_3:
            // No actions in XML

            // Transition to next step: 101
            IF TRUE THEN  // Sequential transition - review XML for actual condition
                #State := STEP_ST10_Flow7_CGlueing_WaitTableCode_OK;
            END_IF;

        // ===========================================
        // STEP 101: WaitTableCode OK
        // ===========================================
        STEP_ST10_Flow7_CGlueing_WaitTableCode_OK:
            // Action Qualifier=N
            // Token: "MES_CHeck_DB".Station_5.CheckStep := 0
            "MES_CHeck_DB".Station_5.CheckStep := 0;
            // Action Qualifier=N
            // Token: "MES_CHeck_DB".Station_5.ResultStep := 0
            "MES_CHeck_DB".Station_5.ResultStep := 0;

            // Transition to next step: 52
            IF TRUE THEN  // Sequential transition - review XML for actual condition
                #State := STEP_ST10_Flow7_CGlueing_Axis_YToGlueePos_6;
            END_IF;

        // ===========================================
        // STEP 52: Axis_YToGlueePos_6
        // ===========================================
        STEP_ST10_Flow7_CGlueing_Axis_YToGlueePos_6:
            // Action Qualifier=N
            // Token: "IAI_DeviceCtl".IAIServo[#Y_axis].Point[4].Start
            "IAI_DeviceCtl".IAIServo[#Y_axis].Point[4].Start;

            // Transition to next step: 85
            IF TRUE THEN  // Sequential transition - review XML for actual condition
                #State := STEP_ST10_Flow7_CGlueing_NGStatus_1;
            END_IF;

        // ===========================================
        // STEP 85: NGStatus_1
        // ===========================================
        STEP_ST10_Flow7_CGlueing_NGStatus_1:
            // Action Qualifier=N
            // Token: "AutoProcessData".C_Glue.PartStatus := 358
            "AutoProcessData".C_Glue.PartStatus := 358;
            // Action Qualifier=N
            // Token: "Station5UnLoadData"."PLC.MagnetIVScore" := "DB_KeyenceCheckerIV3".aDev[1].In.ToolResult[1].nToolMatchingRate
            "Station5UnLoadData"."PLC.MagnetIVScore" := "DB_KeyenceCheckerIV3".aDev[1].In.ToolResult[1].nToolMatchingRate;
            // Action Qualifier=N
            // Token: "AutoProcessData".C_Glue.IV3_MagnetScore := "DB_KeyenceCheckerIV3".aDev[1].In.ToolResult[1].nToolMatchingRate
            "AutoProcessData".C_Glue.IV3_MagnetScore := "DB_KeyenceCheckerIV3".aDev[1].In.ToolResult[1].nToolMatchingRate;
            // Action Qualifier=N
            // Token: "AutoProcessData".C_Glue.IV3_MagnetCheckResult := 2
            "AutoProcessData".C_Glue.IV3_MagnetCheckResult := 2;

            // Transition to next step: 114
            IF TRUE THEN  // Sequential transition - review XML for actual condition
                #State := STEP_ST10_Flow7_CGlueing_GluePos_3;
            END_IF;

        // ===========================================
        // STEP 114: GluePos_3
        // ===========================================
        STEP_ST10_Flow7_CGlueing_GluePos_3:
            // No actions in XML

            // Transition to next step: 146
            IF TRUE THEN  // Sequential transition - review XML for actual condition
                #State := STEP_ST10_Flow7_CGlueing_Step146;
            END_IF;

        // ===========================================
        // STEP 146: Step146
        // ===========================================
        STEP_ST10_Flow7_CGlueing_Step146:
            // No actions in XML

            // Transition to next step: 156
            IF TRUE THEN  // Sequential transition - review XML for actual condition
                #State := STEP_ST10_Flow7_CGlueing_Axis_XYToHomePos_2;
            END_IF;

        // ===========================================
        // STEP 156: Axis_XYToHomePos_2
        // ===========================================
        STEP_ST10_Flow7_CGlueing_Axis_XYToHomePos_2:
            // Action Qualifier=N
            // Token: "IAI_DeviceCtl".IAIServo[#Y_axis].Point[1].Start
            "IAI_DeviceCtl".IAIServo[#Y_axis].Point[1].Start;

            // Transition to next step: 3
            IF TRUE THEN  // Sequential transition - review XML for actual condition
                #State := STEP_ST10_Flow7_CGlueing_S3;
            END_IF;

        // ===========================================
        // STEP 3: S3
        // ===========================================
        STEP_ST10_Flow7_CGlueing_S3:
            // No actions in XML

            // Transition to next step: 113
            IF TRUE THEN  // Sequential transition - review XML for actual condition
                #State := STEP_ST10_Flow7_CGlueing_ServoHomePos_2;
            END_IF;

        // ===========================================
        // STEP 113: ServoHomePos_2
        // ===========================================
        STEP_ST10_Flow7_CGlueing_ServoHomePos_2:
            // Action Qualifier=S
            // Token: "ServoV90_A3".IO.ioAutoHome
            "ServoV90_A3".IO.ioAutoHome := TRUE;

            // Transition to next step: 73
            IF TRUE THEN  // Sequential transition - review XML for actual condition
                #State := STEP_ST10_Flow7_CGlueing_Servo_returns_toGluePos_5;
            END_IF;

        // ===========================================
        // STEP 73: Servo returns toGluePos_5
        // ===========================================
        STEP_ST10_Flow7_CGlueing_Servo_returns_toGluePos_5:
            // Action Qualifier=N
            // Token: "ServoV90_DeviceCtl".V90Servo[3].Point[6].Start
            "ServoV90_DeviceCtl".V90Servo[3].Point[6].Start;

            // Transition to next step: 301
            IF TRUE THEN  // Sequential transition - review XML for actual condition
                #State := STEP_ST10_Flow7_CGlueing_ResetMesCheckRequest;
            END_IF;

        // ===========================================
        // STEP 301: ResetMesCheckRequest
        // ===========================================
        STEP_ST10_Flow7_CGlueing_ResetMesCheckRequest:
            // Action Qualifier=R
            // Token: "PLCtoMES"."PLC.Load_Station5ChickInReq"
            "PLCtoMES"."PLC.Load_Station5ChickInReq" := FALSE;
            // Action Qualifier=R
            // Token: "MEStoPLC"."MES.Load_Station5PartOK"
            "MEStoPLC"."MES.Load_Station5PartOK" := FALSE;
            // Action Qualifier=R
            // Token: "MEStoPLC"."MES.Load_Station5PartNG"
            "MEStoPLC"."MES.Load_Station5PartNG" := FALSE;
            // Action Qualifier=R
            // Token: "MEStoPLC"."MES.Load_Station5ReqMesDone"
            "MEStoPLC"."MES.Load_Station5ReqMesDone" := FALSE;

            // Transition to next step: 79
            IF TRUE THEN  // Sequential transition - review XML for actual condition
                #State := STEP_ST10_Flow7_CGlueing_Axis_XYIVCheckPos;
            END_IF;

        // ===========================================
        // STEP 79: Axis_XYIVCheckPos
        // ===========================================
        STEP_ST10_Flow7_CGlueing_Axis_XYIVCheckPos:
            // Action Qualifier=N
            // Token: "IAI_DeviceCtl".IAIServo[#X_Axis].Point[8].Start
            "IAI_DeviceCtl".IAIServo[#X_Axis].Point[8].Start;

            // Transition to next step: 62
            IF TRUE THEN  // Sequential transition - review XML for actual condition
                #State := STEP_ST10_Flow7_CGlueing_OKStatus;
            END_IF;

        // ===========================================
        // STEP 62: OKStatus
        // ===========================================
        STEP_ST10_Flow7_CGlueing_OKStatus:
            // Action Qualifier=N
            // Token: "AutoProcessData".C_Glue.PartStatus := 310
            "AutoProcessData".C_Glue.PartStatus := 310;
            // Action Qualifier=N
            // Token: "Station5UnLoadData"."PLC.ShaftGlueIVScore1" := "DB_KeyenceCheckerIV3".aDev[2].In.ToolResult[2].nToolMatchingRate
            "Station5UnLoadData"."PLC.ShaftGlueIVScore1" := "DB_KeyenceCheckerIV3".aDev[2].In.ToolResult[2].nToolMatchingRate;
            // Action Qualifier=N
            // Token: "AutoProcessData".C_Glue.IV3_ShaftScore_1 := "DB_KeyenceCheckerIV3".aDev[2].In.ToolResult[2].nToolMatchingRate
            "AutoProcessData".C_Glue.IV3_ShaftScore_1 := "DB_KeyenceCheckerIV3".aDev[2].In.ToolResult[2].nToolMatchingRate;

            // Transition to next step: 5
            IF TRUE THEN  // Sequential transition - review XML for actual condition
                #State := STEP_ST10_Flow7_CGlueing_S5_MESInitial;
            END_IF;

        // ===========================================
        // STEP 5: S5_MESInitial
        // ===========================================
        STEP_ST10_Flow7_CGlueing_S5_MESInitial:
            // No actions in XML

            // Transition to next step: 200
            IF TRUE THEN  // Sequential transition - review XML for actual condition
                #State := STEP_ST10_Flow7_CGlueing_ShaftGluingProcess;
            END_IF;

        // ===========================================
        // STEP 200: ShaftGluingProcess
        // ===========================================
        STEP_ST10_Flow7_CGlueing_ShaftGluingProcess:
            // No actions in XML

            // Transition to next step: 53
            IF TRUE THEN  // Sequential transition - review XML for actual condition
                #State := STEP_ST10_Flow7_CGlueing_Axis_ZToGlueePos_4;
            END_IF;

        // ===========================================
        // STEP 53: Axis_ZToGlueePos_4
        // ===========================================
        STEP_ST10_Flow7_CGlueing_Axis_ZToGlueePos_4:
            // Action Qualifier=N
            // Token: "IAI_DeviceCtl".IAIServo[#Z_Axis].Point[5].Start
            "IAI_DeviceCtl".IAIServo[#Z_Axis].Point[5].Start;

            // Transition to next step: 47
            IF TRUE THEN  // Sequential transition - review XML for actual condition
                #State := STEP_ST10_Flow7_CGlueing_CheckGlueSysOK_2;
            END_IF;

        // ===========================================
        // STEP 47: CheckGlueSysOK_2
        // ===========================================
        STEP_ST10_Flow7_CGlueing_CheckGlueSysOK_2:
            // No actions in XML

            // Transition to next step: 300
            IF TRUE THEN  // Sequential transition - review XML for actual condition
                #State := STEP_ST10_Flow7_CGlueing_RobotPutMagnet;
            END_IF;

        // ===========================================
        // STEP 300: RobotPutMagnet
        // ===========================================
        STEP_ST10_Flow7_CGlueing_RobotPutMagnet:
            // No actions in XML

            // Transition to next step: 59
            IF TRUE THEN  // Sequential transition - review XML for actual condition
                #State := STEP_ST10_Flow7_CGlueing_TimeDelay_4;
            END_IF;

        // ===========================================
        // STEP 59: TimeDelay_4
        // ===========================================
        STEP_ST10_Flow7_CGlueing_TimeDelay_4:
            // No actions in XML

            // Transition to next step: 157
            IF TRUE THEN  // Sequential transition - review XML for actual condition
                #State := STEP_ST10_Flow7_CGlueing_Axis_XYIVCheckPos_1;
            END_IF;

        // ===========================================
        // STEP 157: Axis_XYIVCheckPos_1
        // ===========================================
        STEP_ST10_Flow7_CGlueing_Axis_XYIVCheckPos_1:
            // Action Qualifier=N
            // Token: "IAI_DeviceCtl".IAIServo[#Y_axis].Point[7].Start
            "IAI_DeviceCtl".IAIServo[#Y_axis].Point[7].Start;

            // Transition to next step: 75
            IF TRUE THEN  // Sequential transition - review XML for actual condition
                #State := STEP_ST10_Flow7_CGlueing_Axis_YToGluePos_5;
            END_IF;

        // ===========================================
        // STEP 75: Axis_YToGluePos_5
        // ===========================================
        STEP_ST10_Flow7_CGlueing_Axis_YToGluePos_5:
            // Action Qualifier=N
            // Token: "IAI_DeviceCtl".IAIServo[#Y_axis].Point[6].Start
            "IAI_DeviceCtl".IAIServo[#Y_axis].Point[6].Start;

            // Transition to next step: 121
            IF TRUE THEN  // Sequential transition - review XML for actual condition
                #State := STEP_ST10_Flow7_CGlueing_C_LocationCylinderToWP_2;
            END_IF;

        // ===========================================
        // STEP 121: C-LocationCylinderToWP_2
        // ===========================================
        STEP_ST10_Flow7_CGlueing_C_LocationCylinderToWP_2:
            // Action Qualifier=R
            // Token: "ST10Cylinder".Cy[9].Inout.AutoGoHome
            "ST10Cylinder".Cy[9].Inout.AutoGoHome := FALSE;
            // Action Qualifier=S
            // Token: "ST10Cylinder".Cy[9].Inout.AutoGoWork
            "ST10Cylinder".Cy[9].Inout.AutoGoWork := TRUE;
            // Action Qualifier=R
            // Token: #ioPM_Inface.ProcessComplete
            #ioPM_Inface.ProcessComplete := FALSE;
            // Action Qualifier=S
            // Token: #ioPM_Inface.ProcessStart
            #ioPM_Inface.ProcessStart := TRUE;

            // Transition to next step: 117
            IF TRUE THEN  // Sequential transition - review XML for actual condition
                #State := STEP_ST10_Flow7_CGlueing_ServoHomePos_4;
            END_IF;

        // ===========================================
        // STEP 117: ServoHomePos_4
        // ===========================================
        STEP_ST10_Flow7_CGlueing_ServoHomePos_4:
            // Action Qualifier=S
            // Token: "ServoV90_A3".IO.ioAutoHome
            "ServoV90_A3".IO.ioAutoHome := TRUE;

            // Transition to next step: 31
            IF TRUE THEN  // Sequential transition - review XML for actual condition
                #State := STEP_ST10_Flow7_CGlueing_Servo_returns_toGluePos_1;
            END_IF;

        // ===========================================
        // STEP 31: Servo returns toGluePos_1
        // ===========================================
        STEP_ST10_Flow7_CGlueing_Servo_returns_toGluePos_1:
            // Action Qualifier=N
            // Token: "ServoV90_DeviceCtl".V90Servo[3].Point[2].Start
            "ServoV90_DeviceCtl".V90Servo[3].Point[2].Start;

            // Transition to next step: 100
            IF TRUE THEN  // Sequential transition - review XML for actual condition
                #State := STEP_ST10_Flow7_CGlueing_ProcessStart;
            END_IF;

        // ===========================================
        // STEP 100: ProcessStart
        // ===========================================
        STEP_ST10_Flow7_CGlueing_ProcessStart:
            // Action Qualifier=R
            // Token: #ioPM_Inface.InitialRun
            #ioPM_Inface.InitialRun := FALSE;
            // Action Qualifier=R
            // Token: #ioPM_Inface.ProcessComplete
            #ioPM_Inface.ProcessComplete := FALSE;
            // Action Qualifier=R
            // Token: #ioPM_Inface.ProcessStart
            #ioPM_Inface.ProcessStart := FALSE;
            // Action Qualifier=S
            // Token: #ioPM_Inface.InitialOK
            #ioPM_Inface.InitialOK := TRUE;
            // Action Qualifier=S
            // Token: #ioPM_Inface.WaitRunning
            #ioPM_Inface.WaitRunning := TRUE;
            // Action Qualifier=N, Event="S1"
            // Token: #ioPM_Inface.ProcessResult := 0
            #ioPM_Inface.ProcessResult := 0;
            // Action Qualifier=R
            // Token: "ST10_GeneralData".FlowControl_Handshake[7].Start
            "ST10_GeneralData".FlowControl_Handshake[7].Start := FALSE;
            // Action Qualifier=R
            // Token: "ST10_GeneralData".FlowControl_Handshake[7].Done
            "ST10_GeneralData".FlowControl_Handshake[7].Done := FALSE;

            // Transition to next step: 132
            IF TRUE THEN  // Sequential transition - review XML for actual condition
                #State := STEP_ST10_Flow7_CGlueing_Servo_returns_toGluePos_7;
            END_IF;

        // ===========================================
        // STEP 132: Servo returns toGluePos_7
        // ===========================================
        STEP_ST10_Flow7_CGlueing_Servo_returns_toGluePos_7:
            // Action Qualifier=N
            // Token: "ServoV90_DeviceCtl".V90Servo[3].Point[8].Start
            "ServoV90_DeviceCtl".V90Servo[3].Point[8].Start;

            // Transition to next step: 39
            IF TRUE THEN  // Sequential transition - review XML for actual condition
                #State := STEP_ST10_Flow7_CGlueing_Axis_XToGlueSafPos_2;
            END_IF;

